gfCNCPoint1[3633] = {X 302.1122, Y 47.7433, Z -1.3333, A 0.000, B 0.000, C 0.000 }
gfCNCPoint1[3634] = {X 301.5880, Y 46.9091, Z -1.3333, A 0.000, B 0.000, C 0.000 }
gfCNCPoint1[3635] = {X 301.2626, Y 45.9790, Z -1.3333, A 0.000, B 0.000, C 0.000 }
gfCNCPoint1[3636] = {X 301.1523, Y 44.9999, Z -1.3333, A 0.000, B 0.000, C 0.000 }
gfCNCPoint1[3637] = {X 301.1524, Y 44.1991, Z -1.3333, A 0.000, B 0.000, C 0.000 }
gfCNCPoint1[3638] = {X 301.2707, Y 43.2557, Z -1.3333, A 0.000, B 0.000, C 0.000 }
gfCNCPoint1[3639] = {X 301.5741, Y 42.3546, Z -1.3333, A 0.000, B 0.000, C 0.000 }
gfCNCPoint1[3640] = {X 302.0506, Y 41.5318, Z -1.3333, A 0.000, B 0.000, C 0.000 }
gfCNCPoint1[3641] = {X 302.6811, Y 40.8202, Z -1.3333, A 0.000, B 0.000, C 0.000 }
gfCNCPoint1[3642] = {X 302.6811, Y 34.1143, Z -1.3333, A 0.000, B 0.000, C 0.000 }
gfCNCPoint1[3643] = {X 293.9335, Y 34.1143, Z -1.3333, A 0.000, B 0.000, C 0.000 }
gfCNCPoint1[3644] = {X 293.9325, Y 40.8666, Z -1.3333, A 0.000, B 0.000, C 0.000 }
gfCNCPoint1[3645] = {X 294.5724, Y 41.5615, Z -1.3333, A 0.000, B 0.000, C 0.000 }
gfCNCPoint1[3646] = {X 295.0533, Y 42.3747, Z -1.3333, A 0.000, B 0.000, C 0.000 }
gfCNCPoint1[3647] = {X 295.3539, Y 43.2703, Z -1.3333, A 0.000, B 0.000, C 0.000 }
gfCNCPoint1[3648] = {X 295.4611, Y 44.2089, Z -1.3333, A 0.000, B 0.000, C 0.000 }
gfCNCPoint1[3649] = {X 295.4611, Y 45.0000, Z -1.3333, A 0.000, B 0.000, C 0.000 }
gfCNCPoint1[3650] = {X 295.3508, Y 45.9791, Z -1.3333, A 0.000, B 0.000, C 0.000 }
gfCNCPoint1[3651] = {X 295.0254, Y 46.9091, Z -1.3333, A 0.000, B 0.000, C 0.000 }
gfCNCPoint1[3652] = {X 294.5012, Y 47.7434, Z -1.3333, A 0.000, B 0.000, C 0.000 }
gfCNCPoint1[3653] = {X 293.8045, Y 48.4401, Z -1.3333, A 0.000, B 0.000, C 0.000 }
gfCNCPoint1[3654] = {X 292.9702, Y 48.9643, Z -1.3333, A 0.000, B 0.000, C 0.000 }
gfCNCPoint1[3655] = {X 292.0402, Y 49.2897, Z -1.3333, A 0.000, B 0.000, C 0.000 }
gfCNCPoint1[3656] = {X 291.0611, Y 49.4000, Z -1.3333, A 0.000, B 0.000, C 0.000 }
gfCNCPoint1[3657] = {X 284.6177, Y 49.4000, Z -1.3333, A 0.000, B 0.000, C 0.000 }
gfCNCPoint1[3658] = {X 283.6386, Y 49.2897, Z -1.3333, A 0.000, B 0.000, C 0.000 }
gfCNCPoint1[3659] = {X 282.7086, Y 48.9643, Z -1.3333, A 0.000, B 0.000, C 0.000 }
gfCNCPoint1[3660] = {X 281.8743, Y 48.4400, Z -1.3333, A 0.000, B 0.000, C 0.000 }
gfCNCPoint1[3661] = {X 281.1776, Y 47.7433, Z -1.3333, A 0.000, B 0.000, C 0.000 }
gfCNCPoint1[3662] = {X 280.6534, Y 46.9091, Z -1.3333, A 0.000, B 0.000, C 0.000 }
gfCNCPoint1[3663] = {X 280.3280, Y 45.9791, Z -1.3333, A 0.000, B 0.000, C 0.000 }
gfCNCPoint1[3664] = {X 280.2177, Y 45.0000, Z -1.3333, A 0.000, B 0.000, C 0.000 }
gfCNCPoint1[3665] = {X 280.2177, Y 44.2065, Z -1.3333, A 0.000, B 0.000, C 0.000 }
gfCNCPoint1[3666] = {X 280.3232, Y 43.2697, Z -1.3333, A 0.000, B 0.000, C 0.000 }
gfCNCPoint1[3667] = {X 280.6235, Y 42.3761, Z -1.3333, A 0.000, B 0.000, C 0.000 }
gfCNCPoint1[3668] = {X 281.1051, Y 41.5657, Z -1.3333, A 0.000, B 0.000, C 0.000 }
gfCNCPoint1[3669] = {X 281.7465, Y 40.8749, Z -1.3333, A 0.000, B 0.000, C 0.000 }
gfCNCPoint1[3670] = {X 281.7461, Y 16.3118, Z -1.3333, A 0.000, B 0.000, C 0.000 }
gfCNCPoint1[3671] = {X 281.1011, Y 15.6226, Z -1.3333, A 0.000, B 0.000, C 0.000 }
gfCNCPoint1[3672] = {X 280.6180, Y 14.8117, Z -1.3333, A 0.000, B 0.000, C 0.000 }
gfCNCPoint1[3673] = {X 280.3189, Y 13.9164, Z -1.3333, A 0.000, B 0.000, C 0.000 }
gfCNCPoint1[3674] = {X 280.2177, Y 12.9779, Z -1.3333, A 0.000, B 0.000, C 0.000 }
gfCNCPoint1[3675] = {X 280.2177, Y 12.1868, Z -1.3333, A 0.000, B 0.000, C 0.000 }
gfCNCPoint1[3676] = {X 280.3280, Y 11.2077, Z -1.3333, A 0.000, B 0.000, C 0.000 }
gfCNCPoint1[3677] = {X 280.6534, Y 10.2777, Z -1.3333, A 0.000, B 0.000, C 0.000 }
gfCNCPoint1[3678] = {X 281.1776, Y 9.4435, Z -1.3333, A 0.000, B 0.000, C 0.000 }
gfCNCPoint1[3679] = {X 281.8743, Y 8.7468, Z -1.3333, A 0.000, B 0.000, C 0.000 }
gfCNCPoint1[3680] = {X 282.7086, Y 8.2226, Z -1.3333, A 0.000, B 0.000, C 0.000 }
gfCNCPoint1[3681] = {X 283.6386, Y 7.8971, Z -1.3333, A 0.000, B 0.000, C 0.000 }
gfCNCPoint1[3682] = {X 284.6177, Y 7.7868, Z -1.3333, A 0.000, B 0.000, C 0.000 }
gfCNCPoint1[3683] = {X 291.0611, Y 7.7868, Z -1.3333, A 0.000, B 0.000, C 0.000 }
gfCNCPoint1[3684] = {X 292.0402, Y 7.8971, Z -1.3333, A 0.000, B 0.000, C 0.000 }
gfCNCPoint1[3685] = {X 292.9702, Y 8.2226, Z -1.3333, A 0.000, B 0.000, C 0.000 }
gfCNCPoint1[3686] = {X 293.8045, Y 8.7468, Z -1.3333, A 0.000, B 0.000, C 0.000 }
gfCNCPoint1[3687] = {X 294.5012, Y 9.4435, Z -1.3333, A 0.000, B 0.000, C 0.000 }
gfCNCPoint1[3688] = {X 295.0254, Y 10.2777, Z -1.3333, A 0.000, B 0.000, C 0.000 }
gfCNCPoint1[3689] = {X 295.3508, Y 11.2077, Z -1.3333, A 0.000, B 0.000, C 0.000 }
gfCNCPoint1[3690] = {X 295.4611, Y 12.1868, Z -1.3333, A 0.000, B 0.000, C 0.000 }
gfCNCPoint1[3691] = {X 295.4609, Y 13.0233, Z -1.3333, A 0.000, B 0.000, C 0.000 }
gfCNCPoint1[3692] = {X 295.3525, Y 13.9497, Z -1.3333, A 0.000, B 0.000, C 0.000 }
gfCNCPoint1[3693] = {X 295.0512, Y 14.8325, Z -1.3333, A 0.000, B 0.000, C 0.000 }
gfCNCPoint1[3694] = {X 294.5707, Y 15.6319, Z -1.3333, A 0.000, B 0.000, C 0.000 }
gfCNCPoint1[3695] = {X 293.9324, Y 16.3121, Z -1.3333, A 0.000, B 0.000, C 0.000 }
gfCNCPoint1[3696] = {X 293.9337, Y 22.1165, Z -1.3333, A 0.000, B 0.000, C 0.000 }
gfCNCPoint1[3697] = {X 302.6799, Y 22.1165, Z -1.3333, A 0.000, B 0.000, C 0.000 }
gfCNCPoint1[3698] = {X 302.6806, Y 16.3117, Z -1.3333, A 0.000, B 0.000, C 0.000 }
gfCNCPoint1[3699] = {X 302.0356, Y 15.6225, Z -1.3333, A 0.000, B 0.000, C 0.000 }
gfCNCPoint1[3700] = {X 301.5525, Y 14.8116, Z -1.3333, A 0.000, B 0.000, C 0.000 }
gfCNCPoint1[3701] = {X 301.2535, Y 13.9164, Z -1.3333, A 0.000, B 0.000, C 0.000 }
gfCNCPoint1[3702] = {X 301.1523, Y 12.9779, Z -1.3333, A 0.000, B 0.000, C 0.000 }
gfCNCPoint1[3703] = {X 301.1523, Y 12.1868, Z -1.3333, A 0.000, B 0.000, C 0.000 }
gfCNCPoint1[3704] = {X 301.2626, Y 11.2077, Z -1.3333, A 0.000, B 0.000, C 0.000 }
gfCNCPoint1[3705] = {X 301.5880, Y 10.2777, Z -1.3333, A 0.000, B 0.000, C 0.000 }
gfCNCPoint1[3706] = {X 302.1122, Y 9.4435, Z -1.3333, A 0.000, B 0.000, C 0.000 }
gfCNCPoint1[3707] = {X 302.8089, Y 8.7468, Z -1.3333, A 0.000, B 0.000, C 0.000 }
gfCNCPoint1[3708] = {X 303.6432, Y 8.2226, Z -1.3333, A 0.000, B 0.000, C 0.000 }
gfCNCPoint1[3709] = {X 304.5732, Y 7.8971, Z -1.3333, A 0.000, B 0.000, C 0.000 }
gfCNCPoint1[3710] = {X 305.5523, Y 7.7868, Z -1.3333, A 0.000, B 0.000, C 0.000 }
gfCNCPoint1[3711] = {X 311.9957, Y 7.7868, Z -1.3333, A 0.000, B 0.000, C 0.000 }
gfCNCPoint1[3712] = {X 312.9748, Y 7.8971, Z -1.3333, A 0.000, B 0.000, C 0.000 }
gfCNCPoint1[3713] = {X 313.9048, Y 8.2226, Z -1.3333, A 0.000, B 0.000, C 0.000 }
gfCNCPoint1[3714] = {X 314.7391, Y 8.7468, Z -1.3333, A 0.000, B 0.000, C 0.000 }
gfCNCPoint1[3715] = {X 315.4358, Y 9.4435, Z -1.3333, A 0.000, B 0.000, C 0.000 }
gfCNCPoint1[3716] = {X 315.9600, Y 10.2777, Z -1.3333, A 0.000, B 0.000, C 0.000 }
gfCNCPoint1[3717] = {X 316.2854, Y 11.2077, Z -1.3333, A 0.000, B 0.000, C 0.000 }
gfCNCPoint1[3718] = {X 316.3957, Y 12.1868, Z -1.3333, A 0.000, B 0.000, C 0.000 }
gfCNCPoint1[3719] = {X 316.3955, Y 13.0233, Z -1.3333, A 0.000, B 0.000, C 0.000 }
gfCNCPoint1[3720] = {X 316.2871, Y 13.9497, Z -1.3333, A 0.000, B 0.000, C 0.000 }
gfCNCPoint1[3721] = {X 315.9859, Y 14.8324, Z -1.3333, A 0.000, B 0.000, C 0.000 }
gfCNCPoint1[3722] = {X 315.5054, Y 15.6318, Z -1.3333, A 0.000, B 0.000, C 0.000 }
gfCNCPoint1[3723] = {X 314.8671, Y 16.3119, Z -1.3333, A 0.000, B 0.000, C 0.000 }
gfCNCPoint1[3724] = {X 314.8669, Y 40.8747, Z -1.3333, A 0.000, B 0.000, C 0.000 }
gfCNCPoint1[3725] = {X 315.5120, Y 41.5639, Z -1.3333, A 0.000, B 0.000, C 0.000 }
gfCNCPoint1[3726] = {X 315.9953, Y 42.3749, Z -1.3333, A 0.000, B 0.000, C 0.000 }
gfCNCPoint1[3727] = {X 316.2945, Y 43.2703, Z -1.3333, A 0.000, B 0.000, C 0.000 }
gfCNCPoint1[3728] = {X 316.3957, Y 44.2089, Z -1.3333, A 0.000, B 0.000, C 0.000 }
gfCNCPoint1[3729] = {X 316.3957, Y 45.0000, Z -1.3333, A 0.000, B 0.000, C 0.000 }
gfCNCPoint1[3730] = {X 316.3190, Y 45.8182, Z -1.3333, A 0.000, B 0.000, C 0.000 }
gfCNCPoint1[3731] = {X 316.0914, Y 46.6079, Z -1.3333, A 0.000, B 0.000, C 0.000 }
gfCNCPoint1[3732] = {X 315.7209, Y 47.3415, Z -1.3333, A 0.000, B 0.000, C 0.000 }
gfCNCPoint1[3733] = {X 315.2205, Y 47.9934, Z -1.3333, A 0.000, B 0.000, C 0.000 }
gfCNCPoint1[3734] = {X 315.5723, Y 48.3200, Z -1.3333, A 0.000, B 0.000, C 0.000 }
gfCNCPoint1[3735] = {X 324.3107, Y 48.3200, Z -1.3333, A 0.000, B 0.000, C 0.000 }
gfCNCPoint1[3736] = {X 325.5555, Y 48.4004, Z -1.3333, A 0.000, B 0.000, C 0.000 }
gfCNCPoint1[3737] = {X 326.7797, Y 48.6402, Z -1.3333, A 0.000, B 0.000, C 0.000 }
gfCNCPoint1[3738] = {X 325.5882, Y 48.0963, Z -1.3333, A 0.000, B 0.000, C 0.000 }
gfCNCPoint1[3739] = {X 324.4810, Y 47.3966, Z -1.3333, A 0.000, B 0.000, C 0.000 }
gfCNCPoint1[3740] = {X 323.4784, Y 46.5538, Z -1.3333, A 0.000, B 0.000, C 0.000 }
gfCNCPoint1[3741] = {X 322.8382, Y 45.9295, Z -1.3333, A 0.000, B 0.000, C 0.000 }
gfCNCPoint1[3742] = {X 322.2180, Y 45.2650, Z -1.3333, A 0.000, B 0.000, C 0.000 }
gfCNCPoint1[3743] = {X 321.6628, Y 44.5452, Z -1.3333, A 0.000, B 0.000, C 0.000 }
gfCNCPoint1[3744] = {X 323.6300, Y 43.1703, Z -1.3333, A 0.000, B 0.000, C 0.000 }
gfCNCPoint1[3745] = {X 323.0063, Y 42.0918, Z -1.3333, A 0.000, B 0.000, C 0.000 }
gfCNCPoint1[3746] = {X 322.5757, Y 40.9227, Z -1.3333, A 0.000, B 0.000, C 0.000 }
gfCNCPoint1[3747] = {X 322.3506, Y 39.6973, Z -1.3333, A 0.000, B 0.000, C 0.000 }
gfCNCPoint1[3748] = {X 322.3379, Y 38.4514, Z -1.3333, A 0.000, B 0.000, C 0.000 }
gfCNCPoint1[3749] = {X 322.5377, Y 37.2217, Z -1.3333, A 0.000, B 0.000, C 0.000 }
gfCNCPoint1[3750] = {X 322.9443, Y 36.0440, Z -1.3333, A 0.000, B 0.000, C 0.000 }
gfCNCPoint1[3751] = {X 323.5458, Y 34.9529, Z -1.3333, A 0.000, B 0.000, C 0.000 }
gfCNCPoint1[3752] = {X 327.7789, Y 28.6234, Z -1.3333, A 0.000, B 0.000, C 0.000 }
gfCNCPoint1[3753] = {X 328.5158, Y 27.6951, Z -1.3333, A 0.000, B 0.000, C 0.000 }
gfCNCPoint1[3754] = {X 329.3935, Y 26.8986, Z -1.3333, A 0.000, B 0.000, C 0.000 }
gfCNCPoint1[3755] = {X 330.3889, Y 26.2552, Z -1.3333, A 0.000, B 0.000, C 0.000 }
gfCNCPoint1[3756] = {X 331.5063, Y 25.7713, Z -1.3333, A 0.000, B 0.000, C 0.000 }
gfCNCPoint1[3757] = {X 332.6887, Y 25.4804, Z -1.3333, A 0.000, B 0.000, C 0.000 }
gfCNCPoint1[3758] = {X 333.9031, Y 25.3907, Z -1.3333, A 0.000, B 0.000, C 0.000 }
gfCNCPoint1[3759] = {X 335.1154, Y 25.5046, Z -1.3333, A 0.000, B 0.000, C 0.000 }
gfCNCPoint1[3760] = {X 336.2918, Y 25.8191, Z -1.3333, A 0.000, B 0.000, C 0.000 }
gfCNCPoint1[3761] = {X 337.3993, Y 26.3252, Z -1.3333, A 0.000, B 0.000, C 0.000 }
gfCNCPoint1[3762] = {X 338.1754, Y 26.8292, Z -1.3333, A 0.000, B 0.000, C 0.000 }
gfCNCPoint1[3763] = {X 338.8813, Y 27.4275, Z -1.3333, A 0.000, B 0.000, C 0.000 }
gfCNCPoint1[3764] = {X 339.5028, Y 28.0267, Z -1.3333, A 0.000, B 0.000, C 0.000 }
gfCNCPoint1[3765] = {X 340.3316, Y 28.9979, Z -1.3333, A 0.000, B 0.000, C 0.000 }
gfCNCPoint1[3766] = {X 340.9780, Y 30.0990, Z -1.3333, A 0.000, B 0.000, C 0.000 }
gfCNCPoint1[3767] = {X 341.4220, Y 31.2960, Z -1.3333, A 0.000, B 0.000, C 0.000 }
gfCNCPoint1[3768] = {X 341.6501, Y 32.5522, Z -1.3333, A 0.000, B 0.000, C 0.000 }
gfCNCPoint1[3769] = {X 341.8439, Y 32.7095, Z -1.3333, A 0.000, B 0.000, C 0.000 }
gfCNCPoint1[3770] = {X 342.0399, Y 32.8640, Z -1.3333, A 0.000, B 0.000, C 0.000 }
gfCNCPoint1[3771] = {X 342.9828, Y 33.4816, Z -1.3333, A 0.000, B 0.000, C 0.000 }
gfCNCPoint1[3772] = {X 344.0063, Y 33.9541, Z -1.3333, A 0.000, B 0.000, C 0.000 }
gfCNCPoint1[3773] = {X 345.0879, Y 34.2712, Z -1.3333, A 0.000, B 0.000, C 0.000 }
gfCNCPoint1[3774] = {X 346.2045, Y 34.4260, Z -1.3333, A 0.000, B 0.000, C 0.000 }
gfCNCPoint1[3775] = {X 347.3316, Y 34.4151, Z -1.3333, A 0.000, B 0.000, C 0.000 }
gfCNCPoint1[3776] = {X 348.3037, Y 34.2892, Z -1.3333, A 0.000, B 0.000, C 0.000 }
gfCNCPoint1[3777] = {X 349.2417, Y 34.0051, Z -1.3333, A 0.000, B 0.000, C 0.000 }
gfCNCPoint1[3778] = {X 350.1202, Y 33.5705, Z -1.3333, A 0.000, B 0.000, C 0.000 }
gfCNCPoint1[3779] = {X 350.9153, Y 32.9973, Z -1.3333, A 0.000, B 0.000, C 0.000 }
gfCNCPoint1[3780] = {X 351.7896, Y 32.1460, Z -1.3333, A 0.000, B 0.000, C 0.000 }
gfCNCPoint1[3781] = {X 352.5466, Y 31.1888, Z -1.3333, A 0.000, B 0.000, C 0.000 }
gfCNCPoint1[3782] = {X 353.1735, Y 30.1418, Z -1.3333, A 0.000, B 0.000, C 0.000 }
gfCNCPoint1[3783] = {X 353.6598, Y 29.0226, Z -1.3333, A 0.000, B 0.000, C 0.000 }
gfCNCPoint1[3784] = {X 353.9974, Y 27.8499, Z -1.3333, A 0.000, B 0.000, C 0.000 }
gfCNCPoint1[3785] = {X 354.2247, Y 26.4401, Z -1.3333, A 0.000, B 0.000, C 0.000 }
gfCNCPoint1[3786] = {X 354.3167, Y 25.0152, Z -1.3333, A 0.000, B 0.000, C 0.000 }
gfCNCPoint1[3787] = {X 354.2727, Y 23.5879, Z -1.3333, A 0.000, B 0.000, C 0.000 }
gfCNCPoint1[3788] = {X 354.0929, Y 22.1713, Z -1.3333, A 0.000, B 0.000, C 0.000 }
gfCNCPoint1[3789] = {X 353.8402, Y 21.0759, Z -1.3333, A 0.000, B 0.000, C 0.000 }
gfCNCPoint1[3790] = {X 353.4535, Y 20.0203, Z -1.3333, A 0.000, B 0.000, C 0.000 }
gfCNCPoint1[3791] = {X 352.9388, Y 19.0209, Z -1.3333, A 0.000, B 0.000, C 0.000 }
gfCNCPoint1[3792] = {X 352.3040, Y 18.0930, Z -1.3333, A 0.000, B 0.000, C 0.000 }
gfCNCPoint1[3793] = {X 351.5370, Y 17.2656, Z -1.3333, A 0.000, B 0.000, C 0.000 }
gfCNCPoint1[3794] = {X 350.6343, Y 16.5887, Z -1.3333, A 0.000, B 0.000, C 0.000 }
gfCNCPoint1[3795] = {X 349.6251, Y 16.0843, Z -1.3333, A 0.000, B 0.000, C 0.000 }
gfCNCPoint1[3796] = {X 348.5419, Y 15.7685, Z -1.3333, A 0.000, B 0.000, C 0.000 }
gfCNCPoint1[3797] = {X 347.1562, Y 15.5979, Z -1.3333, A 0.000, B 0.000, C 0.000 }
gfCNCPoint1[3798] = {X 345.7602, Y 15.6140, Z -1.3333, A 0.000, B 0.000, C 0.000 }
gfCNCPoint1[3799] = {X 344.3788, Y 15.8165, Z -1.3333, A 0.000, B 0.000, C 0.000 }
gfCNCPoint1[3800] = {X 343.0368, Y 16.2017, Z -1.3333, A 0.000, B 0.000, C 0.000 }
gfCNCPoint1[3801] = {X 341.7584, Y 16.7629, Z -1.3333, A 0.000, B 0.000, C 0.000 }
gfCNCPoint1[3802] = {X 341.4307, Y 17.8582, Z -1.3333, A 0.000, B 0.000, C 0.000 }
gfCNCPoint1[3803] = {X 340.9356, Y 18.8888, Z -1.3333, A 0.000, B 0.000, C 0.000 }
gfCNCPoint1[3804] = {X 340.2853, Y 19.8292, Z -1.3333, A 0.000, B 0.000, C 0.000 }
gfCNCPoint1[3805] = {X 345.8671, Y 24.3770, Z -1.3333, A 0.000, B 0.000, C 0.000 }
gfCNCPoint1[3806] = {X 346.4664, Y 25.2140, Z -1.3333, A 0.000, B 0.000, C 0.000 }
gfCNCPoint1[3807] = {X 347.0046, Y 26.0914, Z -1.3333, A 0.000, B 0.000, C 0.000 }
gfCNCPoint1[3808] = {X 347.1188, Y 24.7351, Z -1.3333, A 0.000, B 0.000, C 0.000 }
gfCNCPoint1[3809] = {X 346.9949, Y 23.3798, Z -1.3333, A 0.000, B 0.000, C 0.000 }
gfCNCPoint1[3810] = {X 346.9507, Y 23.1695, Z -1.3333, A 0.000, B 0.000, C 0.000 }
gfCNCPoint1[3811] = {X 346.8823, Y 22.9658, Z -1.3333, A 0.000, B 0.000, C 0.000 }
gfCNCPoint1[3812] = {X 346.3959, Y 23.6867, Z -1.3333, A 0.000, B 0.000, C 0.000 }
gfCNCPoint1[3813] = {X 345.8671, Y 24.3770, Z -1.3333, A 0.000, B 0.000, C 0.000 }
gfCNCPoint1[3814] = {X 344.0065, Y 22.8611, Z -1.3333, A 0.000, B 0.000, C 0.000 }
gfCNCPoint1[3815] = {X 343.3271, Y 23.6263, Z -1.3333, A 0.000, B 0.000, C 0.000 }
gfCNCPoint1[3816] = {X 342.5854, Y 24.3313, Z -1.3333, A 0.000, B 0.000, C 0.000 }
gfCNCPoint1[3817] = {X 342.8589, Y 24.5949, Z -1.3333, A 0.000, B 0.000, C 0.000 }
gfCNCPoint1[3818] = {X 343.9812, Y 25.8617, Z -1.3333, A 0.000, B 0.000, C 0.000 }
gfCNCPoint1[3819] = {X 344.9156, Y 27.2729, Z -1.3333, A 0.000, B 0.000, C 0.000 }
gfCNCPoint1[3820] = {X 345.4672, Y 28.3762, Z -1.3333, A 0.000, B 0.000, C 0.000 }
gfCNCPoint1[3821] = {X 345.9035, Y 29.5300, Z -1.3333, A 0.000, B 0.000, C 0.000 }
gfCNCPoint1[3822] = {X 346.4600, Y 29.6326, Z -1.3333, A 0.000, B 0.000, C 0.000 }
gfCNCPoint1[3823] = {X 347.0258, Y 29.6235, Z -1.3333, A 0.000, B 0.000, C 0.000 }
gfCNCPoint1[3824] = {X 347.4365, Y 29.5578, Z -1.3333, A 0.000, B 0.000, C 0.000 }
gfCNCPoint1[3825] = {X 347.7961, Y 29.3489, Z -1.3333, A 0.000, B 0.000, C 0.000 }
gfCNCPoint1[3826] = {X 348.4760, Y 28.6282, Z -1.3333, A 0.000, B 0.000, C 0.000 }
gfCNCPoint1[3827] = {X 348.9866, Y 27.7791, Z -1.3333, A 0.000, B 0.000, C 0.000 }
gfCNCPoint1[3828] = {X 349.3046, Y 26.8407, Z -1.3333, A 0.000, B 0.000, C 0.000 }
gfCNCPoint1[3829] = {X 349.3384, Y 26.6711, Z -1.3333, A 0.000, B 0.000, C 0.000 }
gfCNCPoint1[3830] = {X 349.3694, Y 26.5010, Z -1.3333, A 0.000, B 0.000, C 0.000 }
gfCNCPoint1[3831] = {X 349.5031, Y 25.3293, Z -1.3333, A 0.000, B 0.000, C 0.000 }
gfCNCPoint1[3832] = {X 349.5003, Y 24.1499, Z -1.3333, A 0.000, B 0.000, C 0.000 }
gfCNCPoint1[3833] = {X 349.3613, Y 22.9788, Z -1.3333, A 0.000, B 0.000, C 0.000 }
gfCNCPoint1[3834] = {X 349.1892, Y 22.2869, Z -1.3333, A 0.000, B 0.000, C 0.000 }
gfCNCPoint1[3835] = {X 348.9038, Y 21.6335, Z -1.3333, A 0.000, B 0.000, C 0.000 }
gfCNCPoint1[3836] = {X 348.5130, Y 21.0371, Z -1.3333, A 0.000, B 0.000, C 0.000 }
gfCNCPoint1[3837] = {X 348.1202, Y 20.6777, Z -1.3333, A 0.000, B 0.000, C 0.000 }
gfCNCPoint1[3838] = {X 347.6258, Y 20.4803, Z -1.3333, A 0.000, B 0.000, C 0.000 }
gfCNCPoint1[3839] = {X 346.5729, Y 20.3819, Z -1.3333, A 0.000, B 0.000, C 0.000 }
gfCNCPoint1[3840] = {X 345.5203, Y 20.4822, Z -1.3333, A 0.000, B 0.000, C 0.000 }
gfCNCPoint1[3841] = {X 344.8330, Y 21.7160, Z -1.3333, A 0.000, B 0.000, C 0.000 }
gfCNCPoint1[3842] = {X 344.0065, Y 22.8611, Z -1.3333, A 0.000, B 0.000, C 0.000 }
gfCNCPoint1[3843] = {X 342.1459, Y 21.3451, Z -1.3333, A 0.000, B 0.000, C 0.000 }
gfCNCPoint1[3844] = {X 341.6015, Y 21.9583, Z -1.3333, A 0.000, B 0.000, C 0.000 }
gfCNCPoint1[3845] = {X 341.0072, Y 22.5232, Z -1.3333, A 0.000, B 0.000, C 0.000 }
gfCNCPoint1[3846] = {X 340.7216, Y 22.7630, Z -1.3333, A 0.000, B 0.000, C 0.000 }
gfCNCPoint1[3847] = {X 340.4270, Y 22.9916, Z -1.3333, A 0.000, B 0.000, C 0.000 }
gfCNCPoint1[3848] = {X 339.6615, Y 23.5549, Z -1.3333, A 0.000, B 0.000, C 0.000 }
gfCNCPoint1[3849] = {X 339.1299, Y 23.9121, Z -1.3333, A 0.000, B 0.000, C 0.000 }
gfCNCPoint1[3850] = {X 338.5759, Y 24.2333, Z -1.3333, A 0.000, B 0.000, C 0.000 }
gfCNCPoint1[3851] = {X 339.6079, Y 24.9035, Z -1.3333, A 0.000, B 0.000, C 0.000 }
gfCNCPoint1[3852] = {X 340.5465, Y 25.6991, Z -1.3333, A 0.000, B 0.000, C 0.000 }
gfCNCPoint1[3853] = {X 341.1848, Y 26.3148, Z -1.3333, A 0.000, B 0.000, C 0.000 }
gfCNCPoint1[3854] = {X 342.1202, Y 27.3792, Z -1.3333, A 0.000, B 0.000, C 0.000 }
gfCNCPoint1[3855] = {X 342.8902, Y 28.5687, Z -1.3333, A 0.000, B 0.000, C 0.000 }
gfCNCPoint1[3856] = {X 343.4783, Y 29.8579, Z -1.3333, A 0.000, B 0.000, C 0.000 }
gfCNCPoint1[3857] = {X 343.8718, Y 31.2192, Z -1.3333, A 0.000, B 0.000, C 0.000 }
gfCNCPoint1[3858] = {X 344.6368, Y 31.6221, Z -1.3333, A 0.000, B 0.000, C 0.000 }
gfCNCPoint1[3859] = {X 345.4575, Y 31.8941, Z -1.3333, A 0.000, B 0.000, C 0.000 }
gfCNCPoint1[3860] = {X 346.3117, Y 32.0279, Z -1.3333, A 0.000, B 0.000, C 0.000 }
gfCNCPoint1[3861] = {X 347.1763, Y 32.0198, Z -1.3333, A 0.000, B 0.000, C 0.000 }
gfCNCPoint1[3862] = {X 347.9605, Y 31.9045, Z -1.3333, A 0.000, B 0.000, C 0.000 }
gfCNCPoint1[3863] = {X 348.6994, Y 31.6174, Z -1.3333, A 0.000, B 0.000, C 0.000 }
gfCNCPoint1[3864] = {X 349.3558, Y 31.1730, Z -1.3333, A 0.000, B 0.000, C 0.000 }
gfCNCPoint1[3865] = {X 350.1556, Y 30.3689, Z -1.3333, A 0.000, B 0.000, C 0.000 }
gfCNCPoint1[3866] = {X 350.8155, Y 29.4466, Z -1.3333, A 0.000, B 0.000, C 0.000 }
gfCNCPoint1[3867] = {X 351.3183, Y 28.4300, Z -1.3333, A 0.000, B 0.000, C 0.000 }
gfCNCPoint1[3868] = {X 351.6509, Y 27.3457, Z -1.3333, A 0.000, B 0.000, C 0.000 }
gfCNCPoint1[3869] = {X 351.8790, Y 25.7632, Z -1.3333, A 0.000, B 0.000, C 0.000 }
gfCNCPoint1[3870] = {X 351.9046, Y 24.1645, Z -1.3333, A 0.000, B 0.000, C 0.000 }
gfCNCPoint1[3871] = {X 351.7272, Y 22.5755, Z -1.3333, A 0.000, B 0.000, C 0.000 }
gfCNCPoint1[3872] = {X 351.4581, Y 21.5045, Z -1.3333, A 0.000, B 0.000, C 0.000 }
gfCNCPoint1[3873] = {X 351.0154, Y 20.4929, Z -1.3333, A 0.000, B 0.000, C 0.000 }
gfCNCPoint1[3874] = {X 350.4112, Y 19.5685, Z -1.3333, A 0.000, B 0.000, C 0.000 }
gfCNCPoint1[3875] = {X 349.7601, Y 18.9037, Z -1.3333, A 0.000, B 0.000, C 0.000 }
gfCNCPoint1[3876] = {X 348.9693, Y 18.4129, Z -1.3333, A 0.000, B 0.000, C 0.000 }
gfCNCPoint1[3877] = {X 348.0845, Y 18.1246, Z -1.3333, A 0.000, B 0.000, C 0.000 }
gfCNCPoint1[3878] = {X 346.9931, Y 17.9926, Z -1.3333, A 0.000, B 0.000, C 0.000 }
gfCNCPoint1[3879] = {X 345.8939, Y 18.0111, Z -1.3333, A 0.000, B 0.000, C 0.000 }
gfCNCPoint1[3880] = {X 344.8076, Y 18.1796, Z -1.3333, A 0.000, B 0.000, C 0.000 }
gfCNCPoint1[3881] = {X 343.7545, Y 18.4950, Z -1.3333, A 0.000, B 0.000, C 0.000 }
gfCNCPoint1[3882] = {X 343.3272, Y 19.5038, Z -1.3333, A 0.000, B 0.000, C 0.000 }
gfCNCPoint1[3883] = {X 342.7888, Y 20.4580, Z -1.3333, A 0.000, B 0.000, C 0.000 }
gfCNCPoint1[3884] = {X 342.1459, Y 21.3451, Z -1.3333, A 0.000, B 0.000, C 0.000 }
gfCNCPoint1[3885] = {X 340.2853, Y 19.8292, Z -1.3333, A 0.000, B 0.000, C 0.000 }
gfCNCPoint1[3886] = {X 339.6794, Y 20.4860, Z -1.3333, A 0.000, B 0.000, C 0.000 }
gfCNCPoint1[3887] = {X 338.9976, Y 21.0636, Z -1.3333, A 0.000, B 0.000, C 0.000 }
gfCNCPoint1[3888] = {X 338.2497, Y 21.6140, Z -1.3333, A 0.000, B 0.000, C 0.000 }
gfCNCPoint1[3889] = {X 337.8538, Y 21.8795, Z -1.3333, A 0.000, B 0.000, C 0.000 }
gfCNCPoint1[3890] = {X 337.4413, Y 22.1185, Z -1.3333, A 0.000, B 0.000, C 0.000 }
gfCNCPoint1[3891] = {X 336.3239, Y 22.6023, Z -1.3333, A 0.000, B 0.000, C 0.000 }
gfCNCPoint1[3892] = {X 335.1415, Y 22.8932, Z -1.3333, A 0.000, B 0.000, C 0.000 }
gfCNCPoint1[3893] = {X 333.9271, Y 22.9829, Z -1.3333, A 0.000, B 0.000, C 0.000 }
gfCNCPoint1[3894] = {X 332.7148, Y 22.8690, Z -1.3333, A 0.000, B 0.000, C 0.000 }
gfCNCPoint1[3895] = {X 331.5384, Y 22.5546, Z -1.3333, A 0.000, B 0.000, C 0.000 }
gfCNCPoint1[3896] = {X 330.4309, Y 22.0485, Z -1.3333, A 0.000, B 0.000, C 0.000 }
gfCNCPoint1[3897] = {X 329.5143, Y 21.4374, Z -1.3333, A 0.000, B 0.000, C 0.000 }
gfCNCPoint1[3898] = {X 328.7005, Y 20.6949, Z -1.3333, A 0.000, B 0.000, C 0.000 }
gfCNCPoint1[3899] = {X 328.0080, Y 19.8382, Z -1.3333, A 0.000, B 0.000, C 0.000 }
gfCNCPoint1[3900] = {X 327.4527, Y 18.8868, Z -1.3333, A 0.000, B 0.000, C 0.000 }
gfCNCPoint1[3901] = {X 323.9321, Y 11.6443, Z -1.3333, A 0.000, B 0.000, C 0.000 }
gfCNCPoint1[3902] = {X 323.5337, Y 10.6422, Z -1.3333, A 0.000, B 0.000, C 0.000 }
gfCNCPoint1[3903] = {X 323.2878, Y 9.5922, Z -1.3333, A 0.000, B 0.000, C 0.000 }
gfCNCPoint1[3904] = {X 323.1997, Y 8.5174, Z -1.3333, A 0.000, B 0.000, C 0.000 }
gfCNCPoint1[3905] = {X 323.2713, Y 7.4414, Z -1.3333, A 0.000, B 0.000, C 0.000 }
gfCNCPoint1[3906] = {X 323.4719, Y 6.4885, Z -1.3333, A 0.000, B 0.000, C 0.000 }
gfCNCPoint1[3907] = {X 323.7979, Y 5.5710, Z -1.3333, A 0.000, B 0.000, C 0.000 }
gfCNCPoint1[3908] = {X 324.2435, Y 4.7051, Z -1.3333, A 0.000, B 0.000, C 0.000 }
gfCNCPoint1[3909] = {X 168.0205, Y 4.7051, Z -1.3333, A 0.000, B 0.000, C 0.000 }
gfCNCPoint1[3910] = {X 168.0205, Y 9.5051, Z -1.3333, A 0.000, B 0.000, C 0.000 }
gfCNCPoint1[3911] = {X 166.5360, Y 9.5051, Z -1.3333, A 0.000, B 0.000, C 0.000 }
gfCNCPoint1[3912] = {X 166.5856, Y 9.9932, Z -1.3333, A 0.000, B 0.000, C 0.000 }
gfCNCPoint1[3913] = {X 166.6021, Y 10.4835, Z -1.3333, A 0.000, B 0.000, C 0.000 }
gfCNCPoint1[3914] = {X 166.6021, Y 13.0969, Z -1.3333, A 0.000, B 0.000, C 0.000 }
gfCNCPoint1[3915] = {X 166.8569, Y 11.8210, Z -1.3333, A 0.000, B 0.000, C 0.000 }
gfCNCPoint1[3916] = {X 167.3348, Y 10.6109, Z -1.3333, A 0.000, B 0.000, C 0.000 }
gfCNCPoint1[3917] = {X 168.0205, Y 9.5051, Z -1.3333, A 0.000, B 0.000, C 0.000 }
gfCNCPoint1[3918] = {X 168.0205, Y 7.1051, Z -1.3333, A 0.000, B 0.000, C 0.000 }
gfCNCPoint1[3919] = {X 162.8436, Y 7.1051, Z -1.3333, A 0.000, B 0.000, C 0.000 }
gfCNCPoint1[3920] = {X 163.4703, Y 7.9132, Z -1.3333, A 0.000, B 0.000, C 0.000 }
gfCNCPoint1[3921] = {X 163.9149, Y 8.8342, Z -1.3333, A 0.000, B 0.000, C 0.000 }
gfCNCPoint1[3922] = {X 164.1578, Y 9.8277, Z -1.3333, A 0.000, B 0.000, C 0.000 }
gfCNCPoint1[3923] = {X 164.1910, Y 10.1548, Z -1.3333, A 0.000, B 0.000, C 0.000 }
gfCNCPoint1[3924] = {X 164.2021, Y 10.4835, Z -1.3333, A 0.000, B 0.000, C 0.000 }
gfCNCPoint1[3925] = {X 164.2021, Y 17.4615, Z -1.3333, A 0.000, B 0.000, C 0.000 }
gfCNCPoint1[3926] = {X 164.1140, Y 18.3848, Z -1.3333, A 0.000, B 0.000, C 0.000 }
gfCNCPoint1[3927] = {X 163.8527, Y 19.2747, Z -1.3333, A 0.000, B 0.000, C 0.000 }
gfCNCPoint1[3928] = {X 163.4279, Y 20.0991, Z -1.3333, A 0.000, B 0.000, C 0.000 }
gfCNCPoint1[3929] = {X 162.8547, Y 20.8282, Z -1.3333, A 0.000, B 0.000, C 0.000 }
gfCNCPoint1[3930] = {X 162.1540, Y 21.4358, Z -1.3333, A 0.000, B 0.000, C 0.000 }
gfCNCPoint1[3931] = {X 161.3510, Y 21.8998, Z -1.3333, A 0.000, B 0.000, C 0.000 }
gfCNCPoint1[3932] = {X 160.4746, Y 22.2035, Z -1.3333, A 0.000, B 0.000, C 0.000 }
gfCNCPoint1[3933] = {X 162.1751, Y 29.1998, Z -1.3333, A 0.000, B 0.000, C 0.000 }
gfCNCPoint1[3934] = {X 161.1121, Y 29.4082, Z -1.3333, A 0.000, B 0.000, C 0.000 }
gfCNCPoint1[3935] = {X 160.0347, Y 29.5205, Z -1.3333, A 0.000, B 0.000, C 0.000 }
gfCNCPoint1[3936] = {X 160.0340, Y 38.3367, Z -1.3333, A 0.000, B 0.000, C 0.000 }
gfCNCPoint1[3937] = {X 160.6822, Y 39.6937, Z -1.3333, A 0.000, B 0.000, C 0.000 }
gfCNCPoint1[3938] = {X 161.1574, Y 41.1206, Z -1.3333, A 0.000, B 0.000, C 0.000 }
gfCNCPoint1[3939] = {X 162.0490, Y 41.1205, Z -1.3333, A 0.000, B 0.000, C 0.000 }
gfCNCPoint1[3940] = {X 161.6748, Y 39.3712, Z -1.3333, A 0.000, B 0.000, C 0.000 }
gfCNCPoint1[3941] = {X 161.4508, Y 37.5963, Z -1.3333, A 0.000, B 0.000, C 0.000 }
gfCNCPoint1[3942] = {X 161.3323, Y 35.4809, Z -1.3333, A 0.000, B 0.000, C 0.000 }
gfCNCPoint1[3943] = {X 161.4144, Y 33.3637, Z -1.3333, A 0.000, B 0.000, C 0.000 }
gfCNCPoint1[3944] = {X 161.6961, Y 31.2637, Z -1.3333, A 0.000, B 0.000, C 0.000 }
gfCNCPoint1[3945] = {X 162.1751, Y 29.1998, Z -1.3333, A 0.000, B 0.000, C 0.000 }
gfCNCPoint1[3946] = {X 161.6083, Y 26.8677, Z -1.3333, A 0.000, B 0.000, C 0.000 }
gfCNCPoint1[3947] = {X 160.4733, Y 27.0728, Z -1.3333, A 0.000, B 0.000, C 0.000 }
gfCNCPoint1[3948] = {X 159.3220, Y 27.1415, Z -1.3333, A 0.000, B 0.000, C 0.000 }
gfCNCPoint1[3949] = {X 158.6670, Y 27.1415, Z -1.3333, A 0.000, B 0.000, C 0.000 }
gfCNCPoint1[3950] = {X 158.1502, Y 27.1259, Z -1.3333, A 0.000, B 0.000, C 0.000 }
gfCNCPoint1[3951] = {X 157.6349, Y 27.0829, Z -1.3333, A 0.000, B 0.000, C 0.000 }
gfCNCPoint1[3952] = {X 157.6339, Y 38.9962, Z -1.3333, A 0.000, B 0.000, C 0.000 }
gfCNCPoint1[3953] = {X 158.2178, Y 40.0485, Z -1.3333, A 0.000, B 0.000, C 0.000 }
gfCNCPoint1[3954] = {X 158.6672, Y 41.1650, Z -1.3333, A 0.000, B 0.000, C 0.000 }
gfCNCPoint1[3955] = {X 158.9752, Y 42.3284, Z -1.3333, A 0.000, B 0.000, C 0.000 }
gfCNCPoint1[3956] = {X 159.1372, Y 43.5209, Z -1.3333, A 0.000, B 0.000, C 0.000 }
gfCNCPoint1[3957] = {X 165.4308, Y 43.5200, Z -1.3333, A 0.000, B 0.000, C 0.000 }
gfCNCPoint1[3958] = {X 164.8373, Y 42.0421, Z -1.3333, A 0.000, B 0.000, C 0.000 }
gfCNCPoint1[3959] = {X 164.3724, Y 40.5189, Z -1.3333, A 0.000, B 0.000, C 0.000 }
gfCNCPoint1[3960] = {X 164.0389, Y 38.9575, Z -1.3333, A 0.000, B 0.000, C 0.000 }
gfCNCPoint1[3961] = {X 163.8406, Y 37.3733, Z -1.3333, A 0.000, B 0.000, C 0.000 }
gfCNCPoint1[3962] = {X 163.7324, Y 35.4786, Z -1.3333, A 0.000, B 0.000, C 0.000 }
gfCNCPoint1[3963] = {X 163.8044, Y 33.5822, Z -1.3333, A 0.000, B 0.000, C 0.000 }
gfCNCPoint1[3964] = {X 164.0559, Y 31.7011, Z -1.3333, A 0.000, B 0.000, C 0.000 }
gfCNCPoint1[3965] = {X 164.4847, Y 29.8524, Z -1.3333, A 0.000, B 0.000, C 0.000 }
gfCNCPoint1[3966] = {X 164.8366, Y 28.7335, Z -1.3333, A 0.000, B 0.000, C 0.000 }
gfCNCPoint1[3967] = {X 165.2535, Y 27.6373, Z -1.3333, A 0.000, B 0.000, C 0.000 }
gfCNCPoint1[3968] = {X 165.8702, Y 26.3065, Z -1.3333, A 0.000, B 0.000, C 0.000 }
gfCNCPoint1[3969] = {X 166.6046, Y 25.0369, Z -1.3333, A 0.000, B 0.000, C 0.000 }
gfCNCPoint1[3970] = {X 167.4506, Y 23.8388, Z -1.3333, A 0.000, B 0.000, C 0.000 }
gfCNCPoint1[3971] = {X 167.1640, Y 23.1367, Z -1.3333, A 0.000, B 0.000, C 0.000 }
gfCNCPoint1[3972] = {X 166.2874, Y 24.1837, Z -1.3333, A 0.000, B 0.000, C 0.000 }
gfCNCPoint1[3973] = {X 165.2722, Y 25.0969, Z -1.3333, A 0.000, B 0.000, C 0.000 }
gfCNCPoint1[3974] = {X 164.1386, Y 25.8582, Z -1.3333, A 0.000, B 0.000, C 0.000 }
gfCNCPoint1[3975] = {X 162.9091, Y 26.4524, Z -1.3333, A 0.000, B 0.000, C 0.000 }
gfCNCPoint1[3976] = {X 161.6083, Y 26.8677, Z -1.3333, A 0.000, B 0.000, C 0.000 }
gfCNCPoint1[3977] = {X 161.0415, Y 24.5356, Z -1.3333, A 0.000, B 0.000, C 0.000 }
gfCNCPoint1[3978] = {X 160.1879, Y 24.6899, Z -1.3333, A 0.000, B 0.000, C 0.000 }
gfCNCPoint1[3979] = {X 159.3220, Y 24.7415, Z -1.3333, A 0.000, B 0.000, C 0.000 }
gfCNCPoint1[3980] = {X 158.6755, Y 24.7415, Z -1.3333, A 0.000, B 0.000, C 0.000 }
gfCNCPoint1[3981] = {X 158.2863, Y 24.7298, Z -1.3333, A 0.000, B 0.000, C 0.000 }
gfCNCPoint1[3982] = {X 157.8982, Y 24.6974, Z -1.3333, A 0.000, B 0.000, C 0.000 }
gfCNCPoint1[3983] = {X 156.9776, Y 24.5357, Z -1.3333, A 0.000, B 0.000, C 0.000 }
gfCNCPoint1[3984] = {X 156.0851, Y 24.2580, Z -1.3333, A 0.000, B 0.000, C 0.000 }
gfCNCPoint1[3985] = {X 155.2352, Y 23.8689, Z -1.3333, A 0.000, B 0.000, C 0.000 }
gfCNCPoint1[3986] = {X 155.2339, Y 39.7517, Z -1.3333, A 0.000, B 0.000, C 0.000 }
gfCNCPoint1[3987] = {X 155.8247, Y 40.6440, Z -1.3333, A 0.000, B 0.000, C 0.000 }
gfCNCPoint1[3988] = {X 156.2792, Y 41.6127, Z -1.3333, A 0.000, B 0.000, C 0.000 }
gfCNCPoint1[3989] = {X 156.5877, Y 42.6374, Z -1.3333, A 0.000, B 0.000, C 0.000 }
gfCNCPoint1[3990] = {X 156.7436, Y 43.6961, Z -1.3333, A 0.000, B 0.000, C 0.000 }
gfCNCPoint1[3991] = {X 156.7578, Y 43.9498, Z -1.3333, A 0.000, B 0.000, C 0.000 }
gfCNCPoint1[3992] = {X 156.7631, Y 44.2039, Z -1.3333, A 0.000, B 0.000, C 0.000 }
gfCNCPoint1[3993] = {X 156.7629, Y 45.0588, Z -1.3333, A 0.000, B 0.000, C 0.000 }
gfCNCPoint1[3994] = {X 156.7352, Y 45.6370, Z -1.3333, A 0.000, B 0.000, C 0.000 }
gfCNCPoint1[3995] = {X 156.6616, Y 46.2112, Z -1.3333, A 0.000, B 0.000, C 0.000 }
gfCNCPoint1[3996] = {X 157.9051, Y 46.0006, Z -1.3333, A 0.000, B 0.000, C 0.000 }
gfCNCPoint1[3997] = {X 159.1638, Y 45.9207, Z -1.3333, A 0.000, B 0.000, C 0.000 }
gfCNCPoint1[3998] = {X 159.2309, Y 45.9202, Z -1.3333, A 0.000, B 0.000, C 0.000 }
gfCNCPoint1[3999] = {X 159.2980, Y 45.9200, Z -1.3333, A 0.000, B 0.000, C 0.000 }
gfCNCPoint1[4000] = {X 169.6843, Y 45.9200, Z -1.3333, A 0.000, B 0.000, C 0.000 }
gfCNCPoint1[4001] = {X 168.9035, Y 44.8481, Z -1.3333, A 0.000, B 0.000, C 0.000 }
gfCNCPoint1[4002] = {X 168.2131, Y 43.7159, Z -1.3333, A 0.000, B 0.000, C 0.000 }
gfCNCPoint1[4003] = {X 167.6176, Y 42.5310, Z -1.3333, A 0.000, B 0.000, C 0.000 }
gfCNCPoint1[4004] = {X 166.9496, Y 40.7947, Z -1.3333, A 0.000, B 0.000, C 0.000 }
gfCNCPoint1[4005] = {X 166.4851, Y 38.9932, Z -1.3333, A 0.000, B 0.000, C 0.000 }
gfCNCPoint1[4006] = {X 166.2304, Y 37.1503, Z -1.3333, A 0.000, B 0.000, C 0.000 }
gfCNCPoint1[4007] = {X 166.1319, Y 35.3980, Z -1.3333, A 0.000, B 0.000, C 0.000 }
gfCNCPoint1[4008] = {X 166.2084, Y 33.6446, Z -1.3333, A 0.000, B 0.000, C 0.000 }
gfCNCPoint1[4009] = {X 166.4594, Y 31.9075, Z -1.3333, A 0.000, B 0.000, C 0.000 }
gfCNCPoint1[4010] = {X 166.8822, Y 30.2041, Z -1.3333, A 0.000, B 0.000, C 0.000 }
gfCNCPoint1[4011] = {X 167.4726, Y 28.5514, Z -1.3333, A 0.000, B 0.000, C 0.000 }
gfCNCPoint1[4012] = {X 168.2336, Y 26.9822, Z -1.3333, A 0.000, B 0.000, C 0.000 }
gfCNCPoint1[4013] = {X 169.1861, Y 25.5212, Z -1.3333, A 0.000, B 0.000, C 0.000 }
gfCNCPoint1[4014] = {X 170.3149, Y 24.1918, Z -1.3333, A 0.000, B 0.000, C 0.000 }
gfCNCPoint1[4015] = {X 169.9867, Y 23.6227, Z -1.3333, A 0.000, B 0.000, C 0.000 }
gfCNCPoint1[4016] = {X 169.7113, Y 23.0264, Z -1.3333, A 0.000, B 0.000, C 0.000 }
gfCNCPoint1[4017] = {X 167.1001, Y 16.6309, Z -1.3333, A 0.000, B 0.000, C 0.000 }
gfCNCPoint1[4018] = {X 166.7820, Y 15.6636, Z -1.3333, A 0.000, B 0.000, C 0.000 }
gfCNCPoint1[4019] = {X 166.6021, Y 14.6613, Z -1.3333, A 0.000, B 0.000, C 0.000 }
gfCNCPoint1[4020] = {X 166.6021, Y 17.4615, Z -1.3333, A 0.000, B 0.000, C 0.000 }
gfCNCPoint1[4021] = {X 166.5130, Y 18.5970, Z -1.3333, A 0.000, B 0.000, C 0.000 }
gfCNCPoint1[4022] = {X 166.2479, Y 19.7047, Z -1.3333, A 0.000, B 0.000, C 0.000 }
gfCNCPoint1[4023] = {X 165.8132, Y 20.7575, Z -1.3333, A 0.000, B 0.000, C 0.000 }
gfCNCPoint1[4024] = {X 165.2197, Y 21.7296, Z -1.3333, A 0.000, B 0.000, C 0.000 }
gfCNCPoint1[4025] = {X 164.3788, Y 22.6987, Z -1.3333, A 0.000, B 0.000, C 0.000 }
gfCNCPoint1[4026] = {X 163.3808, Y 23.5052, Z -1.3333, A 0.000, B 0.000, C 0.000 }
gfCNCPoint1[4027] = {X 162.2567, Y 24.1238, Z -1.3333, A 0.000, B 0.000, C 0.000 }
gfCNCPoint1[4028] = {X 161.0415, Y 24.5356, Z -1.3333, A 0.000, B 0.000, C 0.000 }
gfCNCPoint1[4029] = {X 160.4746, Y 22.2035, Z -1.3333, A 0.000, B 0.000, C 0.000 }
gfCNCPoint1[4030] = {X 159.9025, Y 22.3069, Z -1.3333, A 0.000, B 0.000, C 0.000 }
gfCNCPoint1[4031] = {X 159.3220, Y 22.3415, Z -1.3333, A 0.000, B 0.000, C 0.000 }
gfCNCPoint1[4032] = {X 158.6806, Y 22.3415, Z -1.3333, A 0.000, B 0.000, C 0.000 }
gfCNCPoint1[4033] = {X 157.8823, Y 22.2729, Z -1.3333, A 0.000, B 0.000, C 0.000 }
gfCNCPoint1[4034] = {X 157.1058, Y 22.0757, Z -1.3333, A 0.000, B 0.000, C 0.000 }
gfCNCPoint1[4035] = {X 156.3716, Y 21.7550, Z -1.3333, A 0.000, B 0.000, C 0.000 }
gfCNCPoint1[4036] = {X 155.5230, Y 21.1772, Z -1.3333, A 0.000, B 0.000, C 0.000 }
gfCNCPoint1[4037] = {X 154.8127, Y 20.4358, Z -1.3333, A 0.000, B 0.000, C 0.000 }
gfCNCPoint1[4038] = {X 152.8355, Y 20.4368, Z -1.3333, A 0.000, B 0.000, C 0.000 }
gfCNCPoint1[4039] = {X 152.8338, Y 40.6542, Z -1.3333, A 0.000, B 0.000, C 0.000 }
gfCNCPoint1[4040] = {X 153.1758, Y 41.0241, Z -1.3333, A 0.000, B 0.000, C 0.000 }
gfCNCPoint1[4041] = {X 153.6800, Y 41.7287, Z -1.3333, A 0.000, B 0.000, C 0.000 }
gfCNCPoint1[4042] = {X 154.0530, Y 42.5108, Z -1.3333, A 0.000, B 0.000, C 0.000 }
gfCNCPoint1[4043] = {X 154.2830, Y 43.3462, Z -1.3333, A 0.000, B 0.000, C 0.000 }
gfCNCPoint1[4044] = {X 154.3631, Y 44.2089, Z -1.3333, A 0.000, B 0.000, C 0.000 }
gfCNCPoint1[4045] = {X 154.3629, Y 45.0469, Z -1.3333, A 0.000, B 0.000, C 0.000 }
gfCNCPoint1[4046] = {X 154.3440, Y 45.4308, Z -1.3333, A 0.000, B 0.000, C 0.000 }
gfCNCPoint1[4047] = {X 154.2951, Y 45.8119, Z -1.3333, A 0.000, B 0.000, C 0.000 }
gfCNCPoint1[4048] = {X 154.0370, Y 46.7541, Z -1.3333, A 0.000, B 0.000, C 0.000 }
gfCNCPoint1[4049] = {X 153.5963, Y 47.6260, Z -1.3333, A 0.000, B 0.000, C 0.000 }
gfCNCPoint1[4050] = {X 152.9909, Y 48.3926, Z -1.3333, A 0.000, B 0.000, C 0.000 }
gfCNCPoint1[4051] = {X 152.2448, Y 49.0233, Z -1.3333, A 0.000, B 0.000, C 0.000 }
gfCNCPoint1[4052] = {X 151.3881, Y 49.4928, Z -1.3333, A 0.000, B 0.000, C 0.000 }
gfCNCPoint1[4053] = {X 150.4551, Y 49.7822, Z -1.3333, A 0.000, B 0.000, C 0.000 }
gfCNCPoint1[4054] = {X 149.4831, Y 49.8800, Z -1.3333, A 0.000, B 0.000, C 0.000 }
gfCNCPoint1[4055] = {X 143.0396, Y 49.8800, Z -1.3333, A 0.000, B 0.000, C 0.000 }
gfCNCPoint1[4056] = {X 142.0923, Y 49.7872, Z -1.3333, A 0.000, B 0.000, C 0.000 }
gfCNCPoint1[4057] = {X 141.1811, Y 49.5122, Z -1.3333, A 0.000, B 0.000, C 0.000 }
gfCNCPoint1[4058] = {X 140.3405, Y 49.0656, Z -1.3333, A 0.000, B 0.000, C 0.000 }
gfCNCPoint1[4059] = {X 139.6026, Y 48.4643, Z -1.3333, A 0.000, B 0.000, C 0.000 }
gfCNCPoint1[4060] = {X 138.9955, Y 47.7312, Z -1.3333, A 0.000, B 0.000, C 0.000 }
gfCNCPoint1[4061] = {X 138.5423, Y 46.8942, Z -1.3333, A 0.000, B 0.000, C 0.000 }
gfCNCPoint1[4062] = {X 138.2601, Y 45.9852, Z -1.3333, A 0.000, B 0.000, C 0.000 }
gfCNCPoint1[4063] = {X 138.1598, Y 45.0386, Z -1.3333, A 0.000, B 0.000, C 0.000 }
gfCNCPoint1[4064] = {X 138.1601, Y 44.1416, Z -1.3333, A 0.000, B 0.000, C 0.000 }
gfCNCPoint1[4065] = {X 138.2148, Y 43.4769, Z -1.3333, A 0.000, B 0.000, C 0.000 }
gfCNCPoint1[4066] = {X 138.3597, Y 42.8258, Z -1.3333, A 0.000, B 0.000, C 0.000 }
gfCNCPoint1[4067] = {X 129.1532, Y 40.1052, Z -1.3333, A 0.000, B 0.000, C 0.000 }
gfCNCPoint1[4068] = {X 129.5665, Y 38.9035, Z -1.3333, A 0.000, B 0.000, C 0.000 }
gfCNCPoint1[4069] = {X 130.0836, Y 37.7426, Z -1.3333, A 0.000, B 0.000, C 0.000 }
gfCNCPoint1[4070] = {X 130.0836, Y 31.6021, Z -1.3333, A 0.000, B 0.000, C 0.000 }
gfCNCPoint1[4071] = {X 129.2057, Y 31.3795, Z -1.3333, A 0.000, B 0.000, C 0.000 }
gfCNCPoint1[4072] = {X 128.3433, Y 31.1025, Z -1.3333, A 0.000, B 0.000, C 0.000 }
gfCNCPoint1[4073] = {X 128.3430, Y 38.3271, Z -1.3333, A 0.000, B 0.000, C 0.000 }
gfCNCPoint1[4074] = {X 128.7841, Y 39.1998, Z -1.3333, A 0.000, B 0.000, C 0.000 }
gfCNCPoint1[4075] = {X 129.1532, Y 40.1052, Z -1.3333, A 0.000, B 0.000, C 0.000 }
gfCNCPoint1[4076] = {X 131.4548, Y 40.7854, Z -1.3333, A 0.000, B 0.000, C 0.000 }
gfCNCPoint1[4077] = {X 131.9017, Y 39.5320, Z -1.3333, A 0.000, B 0.000, C 0.000 }
gfCNCPoint1[4078] = {X 132.4836, Y 38.3354, Z -1.3333, A 0.000, B 0.000, C 0.000 }
gfCNCPoint1[4079] = {X 132.4836, Y 29.5202, Z -1.3333, A 0.000, B 0.000, C 0.000 }
gfCNCPoint1[4080] = {X 131.3522, Y 29.3993, Z -1.3333, A 0.000, B 0.000, C 0.000 }
gfCNCPoint1[4081] = {X 130.2371, Y 29.1724, Z -1.3333, A 0.000, B 0.000, C 0.000 }
gfCNCPoint1[4082] = {X 129.1484, Y 28.8416, Z -1.3333, A 0.000, B 0.000, C 0.000 }
gfCNCPoint1[4083] = {X 128.0240, Y 28.3761, Z -1.3333, A 0.000, B 0.000, C 0.000 }
gfCNCPoint1[4084] = {X 126.9520, Y 27.7999, Z -1.3333, A 0.000, B 0.000, C 0.000 }
gfCNCPoint1[4085] = {X 125.9435, Y 27.1187, Z -1.3333, A 0.000, B 0.000, C 0.000 }
gfCNCPoint1[4086] = {X 125.9429, Y 38.9879, Z -1.3333, A 0.000, B 0.000, C 0.000 }
gfCNCPoint1[4087] = {X 126.4734, Y 39.9276, Z -1.3333, A 0.000, B 0.000, C 0.000 }
gfCNCPoint1[4088] = {X 126.8960, Y 40.9205, Z -1.3333, A 0.000, B 0.000, C 0.000 }
gfCNCPoint1[4089] = {X 127.2098, Y 41.9730, Z -1.3333, A 0.000, B 0.000, C 0.000 }
gfCNCPoint1[4090] = {X 127.4025, Y 43.0542, Z -1.3333, A 0.000, B 0.000, C 0.000 }
gfCNCPoint1[4091] = {X 127.4714, Y 44.1502, Z -1.3333, A 0.000, B 0.000, C 0.000 }
gfCNCPoint1[4092] = {X 127.4716, Y 45.0000, Z -1.3333, A 0.000, B 0.000, C 0.000 }
gfCNCPoint1[4093] = {X 127.4070, Y 46.1159, Z -1.3333, A 0.000, B 0.000, C 0.000 }
gfCNCPoint1[4094] = {X 127.2143, Y 47.2168, Z -1.3333, A 0.000, B 0.000, C 0.000 }
gfCNCPoint1[4095] = {X 126.8960, Y 48.2883, Z -1.3333, A 0.000, B 0.000, C 0.000 }
gfCNCPoint1[4096] = {X 126.2883, Y 49.6376, Z -1.3333, A 0.000, B 0.000, C 0.000 }
gfCNCPoint1[4097] = {X 125.4821, Y 50.8786, Z -1.3333, A 0.000, B 0.000, C 0.000 }
gfCNCPoint1[4098] = {X 124.4962, Y 51.9821, Z -1.3333, A 0.000, B 0.000, C 0.000 }
gfCNCPoint1[4099] = {X 123.3536, Y 52.9225, Z -1.3333, A 0.000, B 0.000, C 0.000 }
gfCNCPoint1[4100] = {X 122.0810, Y 53.6778, Z -1.3333, A 0.000, B 0.000, C 0.000 }
gfCNCPoint1[4101] = {X 120.7081, Y 54.2302, Z -1.3333, A 0.000, B 0.000, C 0.000 }
gfCNCPoint1[4102] = {X 119.2671, Y 54.5669, Z -1.3333, A 0.000, B 0.000, C 0.000 }
gfCNCPoint1[4103] = {X 117.7916, Y 54.6800, Z -1.3333, A 0.000, B 0.000, C 0.000 }
gfCNCPoint1[4104] = {X 111.9185, Y 54.6800, Z -1.3333, A 0.000, B 0.000, C 0.000 }
gfCNCPoint1[4105] = {X 111.7456, Y 54.6785, Z -1.3333, A 0.000, B 0.000, C 0.000 }
gfCNCPoint1[4106] = {X 111.5728, Y 54.6738, Z -1.3333, A 0.000, B 0.000, C 0.000 }
gfCNCPoint1[4107] = {X 111.0585, Y 69.0646, Z -1.3333, A 0.000, B 0.000, C 0.000 }
gfCNCPoint1[4108] = {X 109.0296, Y 68.9061, Z -1.3333, A 0.000, B 0.000, C 0.000 }
gfCNCPoint1[4109] = {X 107.0213, Y 68.5768, Z -1.3333, A 0.000, B 0.000, C 0.000 }
gfCNCPoint1[4110] = {X 105.0765, Y 68.8983, Z -1.3333, A 0.000, B 0.000, C 0.000 }
gfCNCPoint1[4111] = {X 103.1119, Y 69.0597, Z -1.3333, A 0.000, B 0.000, C 0.000 }
gfCNCPoint1[4112] = {X 101.1407, Y 69.0599, Z -1.3333, A 0.000, B 0.000, C 0.000 }
gfCNCPoint1[4113] = {X 99.1761, Y 68.8989, Z -1.3333, A 0.000, B 0.000, C 0.000 }
gfCNCPoint1[4114] = {X 97.2313, Y 68.5777, Z -1.3333, A 0.000, B 0.000, C 0.000 }
gfCNCPoint1[4115] = {X 95.6131, Y 68.8563, Z -1.3333, A 0.000, B 0.000, C 0.000 }
gfCNCPoint1[4116] = {X 93.9796, Y 69.0240, Z -1.3333, A 0.000, B 0.000, C 0.000 }
gfCNCPoint1[4117] = {X 92.3385, Y 69.0800, Z -1.3333, A 0.000, B 0.000, C 0.000 }
gfCNCPoint1[4118] = {X 86.6884, Y 69.0800, Z -1.3333, A 0.000, B 0.000, C 0.000 }
gfCNCPoint1[4119] = {X 84.7318, Y 70.2668, Z -1.3333, A 0.000, B 0.000, C 0.000 }
gfCNCPoint1[4120] = {X 82.6874, Y 71.2949, Z -1.3333, A 0.000, B 0.000, C 0.000 }
gfCNCPoint1[4121] = {X 107.2717, Y 71.2949, Z -1.3333, A 0.000, B 0.000, C 0.000 }
gfCNCPoint1[4122] = {X 109.1259, Y 70.1132, Z -1.3333, A 0.000, B 0.000, C 0.000 }
gfCNCPoint1[4123] = {X 111.0585, Y 69.0646, Z -1.3333, A 0.000, B 0.000, C 0.000 }
gfCNCPoint1[4124] = {X 111.1442, Y 66.6662, Z -1.3333, A 0.000, B 0.000, C 0.000 }
gfCNCPoint1[4125] = {X 109.0696, Y 66.4920, Z -1.3333, A 0.000, B 0.000, C 0.000 }
gfCNCPoint1[4126] = {X 107.0213, Y 66.1197, Z -1.3333, A 0.000, B 0.000, C 0.000 }
gfCNCPoint1[4127] = {X 105.0796, Y 66.4776, Z -1.3333, A 0.000, B 0.000, C 0.000 }
gfCNCPoint1[4128] = {X 103.1135, Y 66.6574, Z -1.3333, A 0.000, B 0.000, C 0.000 }
gfCNCPoint1[4129] = {X 101.1392, Y 66.6576, Z -1.3333, A 0.000, B 0.000, C 0.000 }
gfCNCPoint1[4130] = {X 99.1730, Y 66.4782, Z -1.3333, A 0.000, B 0.000, C 0.000 }
gfCNCPoint1[4131] = {X 97.2313, Y 66.1207, Z -1.3333, A 0.000, B 0.000, C 0.000 }
gfCNCPoint1[4132] = {X 95.6161, Y 66.4308, Z -1.3333, A 0.000, B 0.000, C 0.000 }
gfCNCPoint1[4133] = {X 93.9821, Y 66.6176, Z -1.3333, A 0.000, B 0.000, C 0.000 }
gfCNCPoint1[4134] = {X 92.3385, Y 66.6800, Z -1.3333, A 0.000, B 0.000, C 0.000 }
gfCNCPoint1[4135] = {X 85.9487, Y 66.6800, Z -1.3333, A 0.000, B 0.000, C 0.000 }
gfCNCPoint1[4136] = {X 83.8781, Y 67.9934, Z -1.3333, A 0.000, B 0.000, C 0.000 }
gfCNCPoint1[4137] = {X 81.6949, Y 69.1097, Z -1.3333, A 0.000, B 0.000, C 0.000 }
gfCNCPoint1[4138] = {X 79.6018, Y 69.9547, Z -1.3333, A 0.000, B 0.000, C 0.000 }
gfCNCPoint1[4139] = {X 77.4444, Y 70.6184, Z -1.3333, A 0.000, B 0.000, C 0.000 }
gfCNCPoint1[4140] = {X 75.2383, Y 71.0959, Z -1.3333, A 0.000, B 0.000, C 0.000 }
gfCNCPoint1[4141] = {X 72.9996, Y 71.3838, Z -1.3333, A 0.000, B 0.000, C 0.000 }
gfCNCPoint1[4142] = {X 70.7445, Y 71.4800, Z -1.3333, A 0.000, B 0.000, C 0.000 }
gfCNCPoint1[4143] = {X 64.1851, Y 71.4800, Z -1.3333, A 0.000, B 0.000, C 0.000 }
gfCNCPoint1[4144] = {X 62.0752, Y 71.3958, Z -1.3333, A 0.000, B 0.000, C 0.000 }
gfCNCPoint1[4145] = {X 59.9787, Y 71.1438, Z -1.3333, A 0.000, B 0.000, C 0.000 }
gfCNCPoint1[4146] = {X 57.9089, Y 70.7255, Z -1.3333, A 0.000, B 0.000, C 0.000 }
gfCNCPoint1[4147] = {X 55.8790, Y 70.1436, Z -1.3333, A 0.000, B 0.000, C 0.000 }
gfCNCPoint1[4148] = {X 53.8492, Y 70.7255, Z -1.3333, A 0.000, B 0.000, C 0.000 }
gfCNCPoint1[4149] = {X 51.7794, Y 71.1438, Z -1.3333, A 0.000, B 0.000, C 0.000 }
gfCNCPoint1[4150] = {X 49.6829, Y 71.3958, Z -1.3333, A 0.000, B 0.000, C 0.000 }
gfCNCPoint1[4151] = {X 47.5729, Y 71.4800, Z -1.3333, A 0.000, B 0.000, C 0.000 }
gfCNCPoint1[4152] = {X 40.6393, Y 71.4800, Z -1.3333, A 0.000, B 0.000, C 0.000 }
gfCNCPoint1[4153] = {X 38.8039, Y 71.4163, Z -1.3333, A 0.000, B 0.000, C 0.000 }
gfCNCPoint1[4154] = {X 36.9773, Y 71.2256, Z -1.3333, A 0.000, B 0.000, C 0.000 }
gfCNCPoint1[4155] = {X 34.3995, Y 72.0336, Z -1.3333, A 0.000, B 0.000, C 0.000 }
gfCNCPoint1[4156] = {X 31.7608, Y 72.6128, Z -1.3333, A 0.000, B 0.000, C 0.000 }
gfCNCPoint1[4157] = {X 30.3286, Y 73.1740, Z -1.3333, A 0.000, B 0.000, C 0.000 }
gfCNCPoint1[4158] = {X 28.8811, Y 73.6949, Z -1.3333, A 0.000, B 0.000, C 0.000 }
gfCNCPoint1[4159] = {X 108.0339, Y 73.6949, Z -1.3333, A 0.000, B 0.000, C 0.000 }
gfCNCPoint1[4160] = {X 110.0295, Y 72.3690, Z -1.3333, A 0.000, B 0.000, C 0.000 }
gfCNCPoint1[4161] = {X 112.1282, Y 71.2131, Z -1.3333, A 0.000, B 0.000, C 0.000 }
gfCNCPoint1[4162] = {X 113.1276, Y 70.7391, Z -1.3333, A 0.000, B 0.000, C 0.000 }
gfCNCPoint1[4163] = {X 114.1445, Y 70.3038, Z -1.3333, A 0.000, B 0.000, C 0.000 }
gfCNCPoint1[4164] = {X 117.4444, Y 66.6800, Z -1.3333, A 0.000, B 0.000, C 0.000 }
gfCNCPoint1[4165] = {X 111.9185, Y 66.6800, Z -1.3333, A 0.000, B 0.000, C 0.000 }
gfCNCPoint1[4166] = {X 111.5313, Y 66.6765, Z -1.3333, A 0.000, B 0.000, C 0.000 }
gfCNCPoint1[4167] = {X 111.1442, Y 66.6662, Z -1.3333, A 0.000, B 0.000, C 0.000 }
gfCNCPoint1[4168] = {X 111.2299, Y 64.2677, Z -1.3333, A 0.000, B 0.000, C 0.000 }
gfCNCPoint1[4169] = {X 109.1084, Y 64.0741, Z -1.3333, A 0.000, B 0.000, C 0.000 }
gfCNCPoint1[4170] = {X 107.0213, Y 63.6477, Z -1.3333, A 0.000, B 0.000, C 0.000 }
gfCNCPoint1[4171] = {X 105.0841, Y 64.0514, Z -1.3333, A 0.000, B 0.000, C 0.000 }
gfCNCPoint1[4172] = {X 103.1158, Y 64.2545, Z -1.3333, A 0.000, B 0.000, C 0.000 }
gfCNCPoint1[4173] = {X 101.1370, Y 64.2547, Z -1.3333, A 0.000, B 0.000, C 0.000 }
gfCNCPoint1[4174] = {X 99.1686, Y 64.0521, Z -1.3333, A 0.000, B 0.000, C 0.000 }
gfCNCPoint1[4175] = {X 97.2313, Y 63.6488, Z -1.3333, A 0.000, B 0.000, C 0.000 }
gfCNCPoint1[4176] = {X 95.6204, Y 63.9986, Z -1.3333, A 0.000, B 0.000, C 0.000 }
gfCNCPoint1[4177] = {X 93.9855, Y 64.2095, Z -1.3333, A 0.000, B 0.000, C 0.000 }
gfCNCPoint1[4178] = {X 92.3385, Y 64.2800, Z -1.3333, A 0.000, B 0.000, C 0.000 }
gfCNCPoint1[4179] = {X 85.8951, Y 64.2800, Z -1.3333, A 0.000, B 0.000, C 0.000 }
gfCNCPoint1[4180] = {X 85.5417, Y 64.2768, Z -1.3333, A 0.000, B 0.000, C 0.000 }
gfCNCPoint1[4181] = {X 85.1884, Y 64.2670, Z -1.3333, A 0.000, B 0.000, C 0.000 }
gfCNCPoint1[4182] = {X 83.3593, Y 65.5113, Z -1.3333, A 0.000, B 0.000, C 0.000 }
gfCNCPoint1[4183] = {X 81.4238, Y 66.5824, Z -1.3333, A 0.000, B 0.000, C 0.000 }
gfCNCPoint1[4184] = {X 79.3981, Y 67.4713, Z -1.3333, A 0.000, B 0.000, C 0.000 }
gfCNCPoint1[4185] = {X 77.2994, Y 68.1706, Z -1.3333, A 0.000, B 0.000, C 0.000 }
gfCNCPoint1[4186] = {X 75.1454, Y 68.6744, Z -1.3333, A 0.000, B 0.000, C 0.000 }
gfCNCPoint1[4187] = {X 72.9543, Y 68.9784, Z -1.3333, A 0.000, B 0.000, C 0.000 }
gfCNCPoint1[4188] = {X 70.7445, Y 69.0800, Z -1.3333, A 0.000, B 0.000, C 0.000 }
gfCNCPoint1[4189] = {X 64.1851, Y 69.0800, Z -1.3333, A 0.000, B 0.000, C 0.000 }
gfCNCPoint1[4190] = {X 62.0678, Y 68.9867, Z -1.3333, A 0.000, B 0.000, C 0.000 }
gfCNCPoint1[4191] = {X 59.9669, Y 68.7076, Z -1.3333, A 0.000, B 0.000, C 0.000 }
gfCNCPoint1[4192] = {X 57.8986, Y 68.2449, Z -1.3333, A 0.000, B 0.000, C 0.000 }
gfCNCPoint1[4193] = {X 55.8790, Y 67.6021, Z -1.3333, A 0.000, B 0.000, C 0.000 }
gfCNCPoint1[4194] = {X 53.8595, Y 68.2449, Z -1.3333, A 0.000, B 0.000, C 0.000 }
gfCNCPoint1[4195] = {X 51.7912, Y 68.7076, Z -1.3333, A 0.000, B 0.000, C 0.000 }
gfCNCPoint1[4196] = {X 49.6903, Y 68.9867, Z -1.3333, A 0.000, B 0.000, C 0.000 }
gfCNCPoint1[4197] = {X 47.5729, Y 69.0800, Z -1.3333, A 0.000, B 0.000, C 0.000 }
gfCNCPoint1[4198] = {X 40.6393, Y 69.0800, Z -1.3333, A 0.000, B 0.000, C 0.000 }
gfCNCPoint1[4199] = {X 38.6735, Y 68.9996, Z -1.3333, A 0.000, B 0.000, C 0.000 }
gfCNCPoint1[4200] = {X 36.7209, Y 68.7591, Z -1.3333, A 0.000, B 0.000, C 0.000 }
gfCNCPoint1[4201] = {X 34.8825, Y 69.3979, Z -1.3333, A 0.000, B 0.000, C 0.000 }
gfCNCPoint1[4202] = {X 33.0046, Y 69.9094, Z -1.3333, A 0.000, B 0.000, C 0.000 }
gfCNCPoint1[4203] = {X 31.0961, Y 70.2912, Z -1.3333, A 0.000, B 0.000, C 0.000 }
gfCNCPoint1[4204] = {X 29.6068, Y 70.8812, Z -1.3333, A 0.000, B 0.000, C 0.000 }
gfCNCPoint1[4205] = {X 28.1002, Y 71.4255, Z -1.3333, A 0.000, B 0.000, C 0.000 }
gfCNCPoint1[4206] = {X 26.8254, Y 71.8460, Z -1.3333, A 0.000, B 0.000, C 0.000 }
gfCNCPoint1[4207] = {X 25.5403, Y 72.2338, Z -1.3333, A 0.000, B 0.000, C 0.000 }
gfCNCPoint1[4208] = {X 24.8758, Y 72.4184, Z -1.3333, A 0.000, B 0.000, C 0.000 }
gfCNCPoint1[4209] = {X 24.3904, Y 72.5501, Z -1.3333, A 0.000, B 0.000, C 0.000 }
gfCNCPoint1[4210] = {X 23.9035, Y 72.6765, Z -1.3333, A 0.000, B 0.000, C 0.000 }
gfCNCPoint1[4211] = {X 23.9035, Y 76.0949, Z -1.3333, A 0.000, B 0.000, C 0.000 }
gfCNCPoint1[4212] = {X 108.8320, Y 76.0949, Z -1.3333, A 0.000, B 0.000, C 0.000 }
gfCNCPoint1[4213] = {X 110.4024, Y 74.9730, Z -1.3333, A 0.000, B 0.000, C 0.000 }
gfCNCPoint1[4214] = {X 112.0503, Y 73.9684, Z -1.3333, A 0.000, B 0.000, C 0.000 }
gfCNCPoint1[4215] = {X 113.7671, Y 73.0865, Z -1.3333, A 0.000, B 0.000, C 0.000 }
gfCNCPoint1[4216] = {X 115.5435, Y 72.3321, Z -1.3333, A 0.000, B 0.000, C 0.000 }
gfCNCPoint1[4217] = {X 123.7293, Y 63.3429, Z -1.3333, A 0.000, B 0.000, C 0.000 }
gfCNCPoint1[4218] = {X 121.7863, Y 63.8616, Z -1.3333, A 0.000, B 0.000, C 0.000 }
gfCNCPoint1[4219] = {X 119.7999, Y 64.1751, Z -1.3333, A 0.000, B 0.000, C 0.000 }
gfCNCPoint1[4220] = {X 117.7916, Y 64.2800, Z -1.3333, A 0.000, B 0.000, C 0.000 }
gfCNCPoint1[4221] = {X 111.9185, Y 64.2800, Z -1.3333, A 0.000, B 0.000, C 0.000 }
gfCNCPoint1[4222] = {X 111.5741, Y 64.2769, Z -1.3333, A 0.000, B 0.000, C 0.000 }
gfCNCPoint1[4223] = {X 111.2299, Y 64.2677, Z -1.3333, A 0.000, B 0.000, C 0.000 }
gfCNCPoint1[4224] = {X 111.3156, Y 61.8692, Z -1.3333, A 0.000, B 0.000, C 0.000 }
gfCNCPoint1[4225] = {X 109.8654, Y 61.7547, Z -1.3333, A 0.000, B 0.000, C 0.000 }
gfCNCPoint1[4226] = {X 108.4304, Y 61.5157, Z -1.3333, A 0.000, B 0.000, C 0.000 }
gfCNCPoint1[4227] = {X 107.0213, Y 61.1540, Z -1.3333, A 0.000, B 0.000, C 0.000 }
gfCNCPoint1[4228] = {X 105.0907, Y 61.6173, Z -1.3333, A 0.000, B 0.000, C 0.000 }
gfCNCPoint1[4229] = {X 103.1191, Y 61.8506, Z -1.3333, A 0.000, B 0.000, C 0.000 }
gfCNCPoint1[4230] = {X 101.1337, Y 61.8509, Z -1.3333, A 0.000, B 0.000, C 0.000 }
gfCNCPoint1[4231] = {X 99.1620, Y 61.6181, Z -1.3333, A 0.000, B 0.000, C 0.000 }
gfCNCPoint1[4232] = {X 97.2313, Y 61.1553, Z -1.3333, A 0.000, B 0.000, C 0.000 }
gfCNCPoint1[4233] = {X 95.6267, Y 61.5566, Z -1.3333, A 0.000, B 0.000, C 0.000 }
gfCNCPoint1[4234] = {X 93.9906, Y 61.7990, Z -1.3333, A 0.000, B 0.000, C 0.000 }
gfCNCPoint1[4235] = {X 92.3385, Y 61.8800, Z -1.3333, A 0.000, B 0.000, C 0.000 }
gfCNCPoint1[4236] = {X 85.8951, Y 61.8800, Z -1.3333, A 0.000, B 0.000, C 0.000 }
gfCNCPoint1[4237] = {X 85.1609, Y 61.8640, Z -1.3333, A 0.000, B 0.000, C 0.000 }
gfCNCPoint1[4238] = {X 84.4280, Y 61.8161, Z -1.3333, A 0.000, B 0.000, C 0.000 }
gfCNCPoint1[4239] = {X 82.7247, Y 63.0692, Z -1.3333, A 0.000, B 0.000, C 0.000 }
gfCNCPoint1[4240] = {X 80.9073, Y 64.1504, Z -1.3333, A 0.000, B 0.000, C 0.000 }
gfCNCPoint1[4241] = {X 78.9932, Y 65.0494, Z -1.3333, A 0.000, B 0.000, C 0.000 }
gfCNCPoint1[4242] = {X 77.0007, Y 65.7577, Z -1.3333, A 0.000, B 0.000, C 0.000 }
gfCNCPoint1[4243] = {X 74.9487, Y 66.2685, Z -1.3333, A 0.000, B 0.000, C 0.000 }
gfCNCPoint1[4244] = {X 72.8566, Y 66.5769, Z -1.3333, A 0.000, B 0.000, C 0.000 }
gfCNCPoint1[4245] = {X 70.7445, Y 66.6800, Z -1.3333, A 0.000, B 0.000, C 0.000 }
gfCNCPoint1[4246] = {X 64.1851, Y 66.6800, Z -1.3333, A 0.000, B 0.000, C 0.000 }
gfCNCPoint1[4247] = {X 62.0576, Y 66.5754, Z -1.3333, A 0.000, B 0.000, C 0.000 }
gfCNCPoint1[4248] = {X 59.9505, Y 66.2624, Z -1.3333, A 0.000, B 0.000, C 0.000 }
gfCNCPoint1[4249] = {X 57.8844, Y 65.7442, Z -1.3333, A 0.000, B 0.000, C 0.000 }
gfCNCPoint1[4250] = {X 55.8790, Y 65.0258, Z -1.3333, A 0.000, B 0.000, C 0.000 }
gfCNCPoint1[4251] = {X 53.8737, Y 65.7442, Z -1.3333, A 0.000, B 0.000, C 0.000 }
gfCNCPoint1[4252] = {X 51.8075, Y 66.2624, Z -1.3333, A 0.000, B 0.000, C 0.000 }
gfCNCPoint1[4253] = {X 49.7005, Y 66.5754, Z -1.3333, A 0.000, B 0.000, C 0.000 }
gfCNCPoint1[4254] = {X 47.5729, Y 66.6800, Z -1.3333, A 0.000, B 0.000, C 0.000 }
gfCNCPoint1[4255] = {X 40.6393, Y 66.6800, Z -1.3333, A 0.000, B 0.000, C 0.000 }
gfCNCPoint1[4256] = {X 38.5438, Y 66.5785, Z -1.3333, A 0.000, B 0.000, C 0.000 }
gfCNCPoint1[4257] = {X 36.4680, Y 66.2749, Z -1.3333, A 0.000, B 0.000, C 0.000 }
gfCNCPoint1[4258] = {X 34.5049, Y 67.0000, Z -1.3333, A 0.000, B 0.000, C 0.000 }
gfCNCPoint1[4259] = {X 32.4899, Y 67.5650, Z -1.3333, A 0.000, B 0.000, C 0.000 }
gfCNCPoint1[4260] = {X 30.4360, Y 67.9662, Z -1.3333, A 0.000, B 0.000, C 0.000 }
gfCNCPoint1[4261] = {X 27.6849, Y 69.0287, Z -1.3333, A 0.000, B 0.000, C 0.000 }
gfCNCPoint1[4262] = {X 24.8761, Y 69.9276, Z -1.3333, A 0.000, B 0.000, C 0.000 }
gfCNCPoint1[4263] = {X 24.2350, Y 70.1056, Z -1.3333, A 0.000, B 0.000, C 0.000 }
gfCNCPoint1[4264] = {X 22.8746, Y 70.4592, Z -1.3333, A 0.000, B 0.000, C 0.000 }
gfCNCPoint1[4265] = {X 21.5035, Y 70.7691, Z -1.3333, A 0.000, B 0.000, C 0.000 }
gfCNCPoint1[4266] = {X 21.5035, Y 78.4949, Z -1.3333, A 0.000, B 0.000, C 0.000 }
gfCNCPoint1[4267] = {X 109.6715, Y 78.4949, Z -1.3333, A 0.000, B 0.000, C 0.000 }
gfCNCPoint1[4268] = {X 111.3433, Y 77.2331, Z -1.3333, A 0.000, B 0.000, C 0.000 }
gfCNCPoint1[4269] = {X 113.1183, Y 76.1214, Z -1.3333, A 0.000, B 0.000, C 0.000 }
gfCNCPoint1[4270] = {X 114.9833, Y 75.1682, Z -1.3333, A 0.000, B 0.000, C 0.000 }
gfCNCPoint1[4271] = {X 116.9240, Y 74.3806, Z -1.3333, A 0.000, B 0.000, C 0.000 }
gfCNCPoint1[4272] = {X 130.4119, Y 59.5691, Z -1.3333, A 0.000, B 0.000, C 0.000 }
gfCNCPoint1[4273] = {X 129.5281, Y 58.7535, Z -1.3333, A 0.000, B 0.000, C 0.000 }
gfCNCPoint1[4274] = {X 128.6970, Y 57.8844, Z -1.3333, A 0.000, B 0.000, C 0.000 }
gfCNCPoint1[4275] = {X 127.3932, Y 58.8832, Z -1.3333, A 0.000, B 0.000, C 0.000 }
gfCNCPoint1[4276] = {X 125.9986, Y 59.7506, Z -1.3333, A 0.000, B 0.000, C 0.000 }
gfCNCPoint1[4277] = {X 124.5262, Y 60.4783, Z -1.3333, A 0.000, B 0.000, C 0.000 }
gfCNCPoint1[4278] = {X 122.9902, Y 61.0595, Z -1.3333, A 0.000, B 0.000, C 0.000 }
gfCNCPoint1[4279] = {X 121.2890, Y 61.5137, Z -1.3333, A 0.000, B 0.000, C 0.000 }
gfCNCPoint1[4280] = {X 119.5499, Y 61.7882, Z -1.3333, A 0.000, B 0.000, C 0.000 }
gfCNCPoint1[4281] = {X 117.7916, Y 61.8800, Z -1.3333, A 0.000, B 0.000, C 0.000 }
gfCNCPoint1[4282] = {X 111.9185, Y 61.8800, Z -1.3333, A 0.000, B 0.000, C 0.000 }
gfCNCPoint1[4283] = {X 111.6170, Y 61.8773, Z -1.3333, A 0.000, B 0.000, C 0.000 }
gfCNCPoint1[4284] = {X 111.3156, Y 61.8692, Z -1.3333, A 0.000, B 0.000, C 0.000 }
gfCNCPoint1[4285] = {X 111.4013, Y 59.4708, Z -1.3333, A 0.000, B 0.000, C 0.000 }
gfCNCPoint1[4286] = {X 109.9149, Y 59.3407, Z -1.3333, A 0.000, B 0.000, C 0.000 }
gfCNCPoint1[4287] = {X 108.4496, Y 59.0584, Z -1.3333, A 0.000, B 0.000, C 0.000 }
gfCNCPoint1[4288] = {X 107.0213, Y 58.6267, Z -1.3333, A 0.000, B 0.000, C 0.000 }
gfCNCPoint1[4289] = {X 105.4260, Y 59.0985, Z -1.3333, A 0.000, B 0.000, C 0.000 }
gfCNCPoint1[4290] = {X 103.7872, Y 59.3842, Z -1.3333, A 0.000, B 0.000, C 0.000 }
gfCNCPoint1[4291] = {X 102.1264, Y 59.4800, Z -1.3333, A 0.000, B 0.000, C 0.000 }
gfCNCPoint1[4292] = {X 100.4656, Y 59.3847, Z -1.3333, A 0.000, B 0.000, C 0.000 }
gfCNCPoint1[4293] = {X 98.8267, Y 59.0996, Z -1.3333, A 0.000, B 0.000, C 0.000 }
gfCNCPoint1[4294] = {X 97.2313, Y 58.6283, Z -1.3333, A 0.000, B 0.000, C 0.000 }
gfCNCPoint1[4295] = {X 95.6367, Y 59.0994, Z -1.3333, A 0.000, B 0.000, C 0.000 }
gfCNCPoint1[4296] = {X 93.9986, Y 59.3845, Z -1.3333, A 0.000, B 0.000, C 0.000 }
gfCNCPoint1[4297] = {X 92.3385, Y 59.4800, Z -1.3333, A 0.000, B 0.000, C 0.000 }
gfCNCPoint1[4298] = {X 85.8951, Y 59.4800, Z -1.3333, A 0.000, B 0.000, C 0.000 }
gfCNCPoint1[4299] = {X 84.7780, Y 59.4368, Z -1.3333, A 0.000, B 0.000, C 0.000 }
gfCNCPoint1[4300] = {X 83.6677, Y 59.3077, Z -1.3333, A 0.000, B 0.000, C 0.000 }
gfCNCPoint1[4301] = {X 82.0978, Y 60.5827, Z -1.3333, A 0.000, B 0.000, C 0.000 }
gfCNCPoint1[4302] = {X 80.4031, Y 61.6862, Z -1.3333, A 0.000, B 0.000, C 0.000 }
gfCNCPoint1[4303] = {X 78.6021, Y 62.6061, Z -1.3333, A 0.000, B 0.000, C 0.000 }
gfCNCPoint1[4304] = {X 76.7146, Y 63.3324, Z -1.3333, A 0.000, B 0.000, C 0.000 }
gfCNCPoint1[4305] = {X 74.7614, Y 63.8569, Z -1.3333, A 0.000, B 0.000, C 0.000 }
gfCNCPoint1[4306] = {X 72.7640, Y 64.1739, Z -1.3333, A 0.000, B 0.000, C 0.000 }
gfCNCPoint1[4307] = {X 70.7445, Y 64.2800, Z -1.3333, A 0.000, B 0.000, C 0.000 }
gfCNCPoint1[4308] = {X 64.1851, Y 64.2800, Z -1.3333, A 0.000, B 0.000, C 0.000 }
gfCNCPoint1[4309] = {X 62.0428, Y 64.1606, Z -1.3333, A 0.000, B 0.000, C 0.000 }
gfCNCPoint1[4310] = {X 59.9269, Y 63.8039, Z -1.3333, A 0.000, B 0.000, C 0.000 }
gfCNCPoint1[4311] = {X 57.8638, Y 63.2143, Z -1.3333, A 0.000, B 0.000, C 0.000 }
gfCNCPoint1[4312] = {X 55.8790, Y 62.3991, Z -1.3333, A 0.000, B 0.000, C 0.000 }
gfCNCPoint1[4313] = {X 53.8942, Y 63.2143, Z -1.3333, A 0.000, B 0.000, C 0.000 }
gfCNCPoint1[4314] = {X 51.8311, Y 63.8039, Z -1.3333, A 0.000, B 0.000, C 0.000 }
gfCNCPoint1[4315] = {X 49.7153, Y 64.1606, Z -1.3333, A 0.000, B 0.000, C 0.000 }
gfCNCPoint1[4316] = {X 47.5729, Y 64.2800, Z -1.3333, A 0.000, B 0.000, C 0.000 }
gfCNCPoint1[4317] = {X 40.6393, Y 64.2800, Z -1.3333, A 0.000, B 0.000, C 0.000 }
gfCNCPoint1[4318] = {X 39.1544, Y 64.2227, Z -1.3333, A 0.000, B 0.000, C 0.000 }
gfCNCPoint1[4319] = {X 37.6782, Y 64.0513, Z -1.3333, A 0.000, B 0.000, C 0.000 }
gfCNCPoint1[4320] = {X 36.2197, Y 63.7666, Z -1.3333, A 0.000, B 0.000, C 0.000 }
gfCNCPoint1[4321] = {X 34.1362, Y 64.5931, Z -1.3333, A 0.000, B 0.000, C 0.000 }
gfCNCPoint1[4322] = {X 31.9837, Y 65.2184, Z -1.3333, A 0.000, B 0.000, C 0.000 }
gfCNCPoint1[4323] = {X 29.7817, Y 65.6368, Z -1.3333, A 0.000, B 0.000, C 0.000 }
gfCNCPoint1[4324] = {X 27.0275, Y 66.7154, Z -1.3333, A 0.000, B 0.000, C 0.000 }
gfCNCPoint1[4325] = {X 24.2118, Y 67.6213, Z -1.3333, A 0.000, B 0.000, C 0.000 }
gfCNCPoint1[4326] = {X 23.5941, Y 67.7927, Z -1.3333, A 0.000, B 0.000, C 0.000 }
gfCNCPoint1[4327] = {X 21.3624, Y 68.3451, Z -1.3333, A 0.000, B 0.000, C 0.000 }
gfCNCPoint1[4328] = {X 19.1035, Y 68.7732, Z -1.3333, A 0.000, B 0.000, C 0.000 }
gfCNCPoint1[4329] = {X 19.1035, Y 80.8949, Z -1.3333, A 0.000, B 0.000, C 0.000 }
gfCNCPoint1[4330] = {X 110.5598, Y 80.8949, Z -1.3333, A 0.000, B 0.000, C 0.000 }
gfCNCPoint1[4331] = {X 112.3074, Y 79.4898, Z -1.3333, A 0.000, B 0.000, C 0.000 }
gfCNCPoint1[4332] = {X 114.1908, Y 78.2728, Z -1.3333, A 0.000, B 0.000, C 0.000 }
gfCNCPoint1[4333] = {X 116.1898, Y 77.2568, Z -1.3333, A 0.000, B 0.000, C 0.000 }
gfCNCPoint1[4334] = {X 118.2831, Y 76.4527, Z -1.3333, A 0.000, B 0.000, C 0.000 }
gfCNCPoint1[4335] = {X 133.9641, Y 59.2327, Z -1.3333, A 0.000, B 0.000, C 0.000 }
gfCNCPoint1[4336] = {X 132.7160, Y 58.3551, Z -1.3333, A 0.000, B 0.000, C 0.000 }
gfCNCPoint1[4337] = {X 131.5523, Y 57.3683, Z -1.3333, A 0.000, B 0.000, C 0.000 }
gfCNCPoint1[4338] = {X 130.4824, Y 56.2805, Z -1.3333, A 0.000, B 0.000, C 0.000 }
gfCNCPoint1[4339] = {X 129.6655, Y 55.2988, Z -1.3333, A 0.000, B 0.000, C 0.000 }
gfCNCPoint1[4340] = {X 128.9251, Y 54.2582, Z -1.3333, A 0.000, B 0.000, C 0.000 }
gfCNCPoint1[4341] = {X 128.0750, Y 55.1942, Z -1.3333, A 0.000, B 0.000, C 0.000 }
gfCNCPoint1[4342] = {X 127.1464, Y 56.0525, Z -1.3333, A 0.000, B 0.000, C 0.000 }
gfCNCPoint1[4343] = {X 125.7915, Y 57.0695, Z -1.3333, A 0.000, B 0.000, C 0.000 }
gfCNCPoint1[4344] = {X 124.3270, Y 57.9212, Z -1.3333, A 0.000, B 0.000, C 0.000 }
gfCNCPoint1[4345] = {X 122.7731, Y 58.5961, Z -1.3333, A 0.000, B 0.000, C 0.000 }
gfCNCPoint1[4346] = {X 121.1510, Y 59.0849, Z -1.3333, A 0.000, B 0.000, C 0.000 }
gfCNCPoint1[4347] = {X 119.4828, Y 59.3809, Z -1.3333, A 0.000, B 0.000, C 0.000 }
gfCNCPoint1[4348] = {X 117.7916, Y 59.4800, Z -1.3333, A 0.000, B 0.000, C 0.000 }
gfCNCPoint1[4349] = {X 111.9185, Y 59.4800, Z -1.3333, A 0.000, B 0.000, C 0.000 }
gfCNCPoint1[4350] = {X 111.6599, Y 59.4777, Z -1.3333, A 0.000, B 0.000, C 0.000 }
gfCNCPoint1[4351] = {X 111.4013, Y 59.4708, Z -1.3333, A 0.000, B 0.000, C 0.000 }
gfCNCPoint1[4352] = {X 111.4871, Y 57.0723, Z -1.3333, A 0.000, B 0.000, C 0.000 }
gfCNCPoint1[4353] = {X 109.9587, Y 56.9200, Z -1.3333, A 0.000, B 0.000, C 0.000 }
gfCNCPoint1[4354] = {X 108.4621, Y 56.5750, Z -1.3333, A 0.000, B 0.000, C 0.000 }
gfCNCPoint1[4355] = {X 107.0213, Y 56.0428, Z -1.3333, A 0.000, B 0.000, C 0.000 }
gfCNCPoint1[4356] = {X 105.4432, Y 56.6151, Z -1.3333, A 0.000, B 0.000, C 0.000 }
gfCNCPoint1[4357] = {X 103.8010, Y 56.9630, Z -1.3333, A 0.000, B 0.000, C 0.000 }
gfCNCPoint1[4358] = {X 102.1265, Y 57.0800, Z -1.3333, A 0.000, B 0.000, C 0.000 }
gfCNCPoint1[4359] = {X 100.4519, Y 56.9637, Z -1.3333, A 0.000, B 0.000, C 0.000 }
gfCNCPoint1[4360] = {X 98.8096, Y 56.6164, Z -1.3333, A 0.000, B 0.000, C 0.000 }
gfCNCPoint1[4361] = {X 97.2313, Y 56.0448, Z -1.3333, A 0.000, B 0.000, C 0.000 }
gfCNCPoint1[4362] = {X 95.6538, Y 56.6162, Z -1.3333, A 0.000, B 0.000, C 0.000 }
gfCNCPoint1[4363] = {X 94.0123, Y 56.9635, Z -1.3333, A 0.000, B 0.000, C 0.000 }
gfCNCPoint1[4364] = {X 92.3385, Y 57.0800, Z -1.3333, A 0.000, B 0.000, C 0.000 }
gfCNCPoint1[4365] = {X 85.8951, Y 57.0800, Z -1.3333, A 0.000, B 0.000, C 0.000 }
gfCNCPoint1[4366] = {X 84.3894, Y 56.9858, Z -1.3333, A 0.000, B 0.000, C 0.000 }
gfCNCPoint1[4367] = {X 82.9073, Y 56.7047, Z -1.3333, A 0.000, B 0.000, C 0.000 }
gfCNCPoint1[4368] = {X 81.4847, Y 58.0224, Z -1.3333, A 0.000, B 0.000, C 0.000 }
gfCNCPoint1[4369] = {X 79.9203, Y 59.1682, Z -1.3333, A 0.000, B 0.000, C 0.000 }
gfCNCPoint1[4370] = {X 78.2348, Y 60.1271, Z -1.3333, A 0.000, B 0.000, C 0.000 }
gfCNCPoint1[4371] = {X 76.4504, Y 60.8864, Z -1.3333, A 0.000, B 0.000, C 0.000 }
gfCNCPoint1[4372] = {X 74.5908, Y 61.4359, Z -1.3333, A 0.000, B 0.000, C 0.000 }
gfCNCPoint1[4373] = {X 72.6804, Y 61.7686, Z -1.3333, A 0.000, B 0.000, C 0.000 }
gfCNCPoint1[4374] = {X 70.7445, Y 61.8800, Z -1.3333, A 0.000, B 0.000, C 0.000 }
gfCNCPoint1[4375] = {X 64.1851, Y 61.8800, Z -1.3333, A 0.000, B 0.000, C 0.000 }
gfCNCPoint1[4376] = {X 62.4514, Y 61.7907, Z -1.3333, A 0.000, B 0.000, C 0.000 }
gfCNCPoint1[4377] = {X 60.7359, Y 61.5238, Z -1.3333, A 0.000, B 0.000, C 0.000 }
gfCNCPoint1[4378] = {X 59.0570, Y 61.0822, Z -1.3333, A 0.000, B 0.000, C 0.000 }
gfCNCPoint1[4379] = {X 57.4323, Y 60.4704, Z -1.3333, A 0.000, B 0.000, C 0.000 }
gfCNCPoint1[4380] = {X 55.8790, Y 59.6950, Z -1.3333, A 0.000, B 0.000, C 0.000 }
gfCNCPoint1[4381] = {X 54.3258, Y 60.4704, Z -1.3333, A 0.000, B 0.000, C 0.000 }
gfCNCPoint1[4382] = {X 52.7011, Y 61.0822, Z -1.3333, A 0.000, B 0.000, C 0.000 }
gfCNCPoint1[4383] = {X 51.0221, Y 61.5238, Z -1.3333, A 0.000, B 0.000, C 0.000 }
gfCNCPoint1[4384] = {X 49.3067, Y 61.7907, Z -1.3333, A 0.000, B 0.000, C 0.000 }
gfCNCPoint1[4385] = {X 47.5729, Y 61.8800, Z -1.3333, A 0.000, B 0.000, C 0.000 }
gfCNCPoint1[4386] = {X 40.6393, Y 61.8800, Z -1.3333, A 0.000, B 0.000, C 0.000 }
gfCNCPoint1[4387] = {X 39.0674, Y 61.8067, Z -1.3333, A 0.000, B 0.000, C 0.000 }
gfCNCPoint1[4388] = {X 37.5092, Y 61.5872, Z -1.3333, A 0.000, B 0.000, C 0.000 }
gfCNCPoint1[4389] = {X 35.9782, Y 61.2237, Z -1.3333, A 0.000, B 0.000, C 0.000 }
gfCNCPoint1[4390] = {X 34.3395, Y 61.9591, Z -1.3333, A 0.000, B 0.000, C 0.000 }
gfCNCPoint1[4391] = {X 32.6445, Y 62.5533, Z -1.3333, A 0.000, B 0.000, C 0.000 }
gfCNCPoint1[4392] = {X 30.9053, Y 63.0020, Z -1.3333, A 0.000, B 0.000, C 0.000 }
gfCNCPoint1[4393] = {X 29.1344, Y 63.3020, Z -1.3333, A 0.000, B 0.000, C 0.000 }
gfCNCPoint1[4394] = {X 26.3794, Y 64.3982, Z -1.3333, A 0.000, B 0.000, C 0.000 }
gfCNCPoint1[4395] = {X 23.5587, Y 65.3119, Z -1.3333, A 0.000, B 0.000, C 0.000 }
gfCNCPoint1[4396] = {X 22.9533, Y 65.4799, Z -1.3333, A 0.000, B 0.000, C 0.000 }
gfCNCPoint1[4397] = {X 20.8927, Y 65.9911, Z -1.3333, A 0.000, B 0.000, C 0.000 }
gfCNCPoint1[4398] = {X 18.8074, Y 66.3898, Z -1.3333, A 0.000, B 0.000, C 0.000 }
gfCNCPoint1[4399] = {X 16.7035, Y 66.6749, Z -1.3333, A 0.000, B 0.000, C 0.000 }
gfCNCPoint1[4400] = {X 16.7035, Y 83.2949, Z -1.3333, A 0.000, B 0.000, C 0.000 }
gfCNCPoint1[4401] = {X 111.5064, Y 83.2949, Z -1.3333, A 0.000, B 0.000, C 0.000 }
gfCNCPoint1[4402] = {X 112.9253, Y 82.0353, Z -1.3333, A 0.000, B 0.000, C 0.000 }
gfCNCPoint1[4403] = {X 114.4611, Y 80.9213, Z -1.3333, A 0.000, B 0.000, C 0.000 }
gfCNCPoint1[4404] = {X 116.0990, Y 79.9636, Z -1.3333, A 0.000, B 0.000, C 0.000 }
gfCNCPoint1[4405] = {X 117.8231, Y 79.1715, Z -1.3333, A 0.000, B 0.000, C 0.000 }
gfCNCPoint1[4406] = {X 119.6167, Y 78.5527, Z -1.3333, A 0.000, B 0.000, C 0.000 }
gfCNCPoint1[4407] = {X 137.8581, Y 58.5212, Z -1.3333, A 0.000, B 0.000, C 0.000 }
gfCNCPoint1[4408] = {X 136.5232, Y 57.9308, Z -1.3333, A 0.000, B 0.000, C 0.000 }
gfCNCPoint1[4409] = {X 135.2545, Y 57.2091, Z -1.3333, A 0.000, B 0.000, C 0.000 }
gfCNCPoint1[4410] = {X 134.0104, Y 56.3200, Z -1.3333, A 0.000, B 0.000, C 0.000 }
gfCNCPoint1[4411] = {X 132.8669, Y 55.3047, Z -1.3333, A 0.000, B 0.000, C 0.000 }
gfCNCPoint1[4412] = {X 131.8370, Y 54.1745, Z -1.3333, A 0.000, B 0.000, C 0.000 }
gfCNCPoint1[4413] = {X 130.9319, Y 52.9419, Z -1.3333, A 0.000, B 0.000, C 0.000 }
gfCNCPoint1[4414] = {X 130.2147, Y 51.7225, Z -1.3333, A 0.000, B 0.000, C 0.000 }
gfCNCPoint1[4415] = {X 129.6199, Y 50.4390, Z -1.3333, A 0.000, B 0.000, C 0.000 }
gfCNCPoint1[4416] = {X 129.1532, Y 49.1035, Z -1.3333, A 0.000, B 0.000, C 0.000 }
gfCNCPoint1[4417] = {X 128.6036, Y 50.3877, Z -1.3333, A 0.000, B 0.000, C 0.000 }
gfCNCPoint1[4418] = {X 127.9093, Y 51.5998, Z -1.3333, A 0.000, B 0.000, C 0.000 }
gfCNCPoint1[4419] = {X 127.0798, Y 52.7237, Z -1.3333, A 0.000, B 0.000, C 0.000 }
gfCNCPoint1[4420] = {X 126.0417, Y 53.8239, Z -1.3333, A 0.000, B 0.000, C 0.000 }
gfCNCPoint1[4421] = {X 124.8743, Y 54.7858, Z -1.3333, A 0.000, B 0.000, C 0.000 }
gfCNCPoint1[4422] = {X 123.5958, Y 55.5942, Z -1.3333, A 0.000, B 0.000, C 0.000 }
gfCNCPoint1[4423] = {X 122.2263, Y 56.2365, Z -1.3333, A 0.000, B 0.000, C 0.000 }
gfCNCPoint1[4424] = {X 120.7872, Y 56.7027, Z -1.3333, A 0.000, B 0.000, C 0.000 }
gfCNCPoint1[4425] = {X 119.3012, Y 56.9853, Z -1.3333, A 0.000, B 0.000, C 0.000 }
gfCNCPoint1[4426] = {X 117.7916, Y 57.0800, Z -1.3333, A 0.000, B 0.000, C 0.000 }
gfCNCPoint1[4427] = {X 111.9185, Y 57.0800, Z -1.3333, A 0.000, B 0.000, C 0.000 }
gfCNCPoint1[4428] = {X 111.7027, Y 57.0781, Z -1.3333, A 0.000, B 0.000, C 0.000 }
gfCNCPoint1[4429] = {X 111.4871, Y 57.0723, Z -1.3333, A 0.000, B 0.000, C 0.000 }
gfCNCPoint1[4430] = {X 111.5728, Y 54.6738, Z -1.3333, A 0.000, B 0.000, C 0.000 }
gfCNCPoint1[4431] = {X 110.3820, Y 54.5573, Z -1.3333, A 0.000, B 0.000, C 0.000 }
gfCNCPoint1[4432] = {X 109.2147, Y 54.2947, Z -1.3333, A 0.000, B 0.000, C 0.000 }
gfCNCPoint1[4433] = {X 108.0887, Y 53.8902, Z -1.3333, A 0.000, B 0.000, C 0.000 }
gfCNCPoint1[4434] = {X 107.0213, Y 53.3498, Z -1.3333, A 0.000, B 0.000, C 0.000 }
gfCNCPoint1[4435] = {X 106.6480, Y 53.5578, Z -1.3333, A 0.000, B 0.000, C 0.000 }
gfCNCPoint1[4436] = {X 106.2658, Y 53.7492, Z -1.3333, A 0.000, B 0.000, C 0.000 }
gfCNCPoint1[4437] = {X 105.0149, Y 54.2383, Z -1.3333, A 0.000, B 0.000, C 0.000 }
gfCNCPoint1[4438] = {X 103.7084, Y 54.5495, Z -1.3333, A 0.000, B 0.000, C 0.000 }
gfCNCPoint1[4439] = {X 102.3713, Y 54.6768, Z -1.3333, A 0.000, B 0.000, C 0.000 }
gfCNCPoint1[4440] = {X 101.0295, Y 54.6179, Z -1.3333, A 0.000, B 0.000, C 0.000 }
gfCNCPoint1[4441] = {X 99.7088, Y 54.3738, Z -1.3333, A 0.000, B 0.000, C 0.000 }
gfCNCPoint1[4442] = {X 98.4345, Y 53.9493, Z -1.3333, A 0.000, B 0.000, C 0.000 }
gfCNCPoint1[4443] = {X 97.2313, Y 53.3524, Z -1.3333, A 0.000, B 0.000, C 0.000 }
gfCNCPoint1[4444] = {X 96.0852, Y 53.9255, Z -1.3333, A 0.000, B 0.000, C 0.000 }
gfCNCPoint1[4445] = {X 94.8734, Y 54.3422, Z -1.3333, A 0.000, B 0.000, C 0.000 }
gfCNCPoint1[4446] = {X 93.6172, Y 54.5952, Z -1.3333, A 0.000, B 0.000, C 0.000 }
gfCNCPoint1[4447] = {X 92.3385, Y 54.6800, Z -1.3333, A 0.000, B 0.000, C 0.000 }
gfCNCPoint1[4448] = {X 85.8951, Y 54.6800, Z -1.3333, A 0.000, B 0.000, C 0.000 }
gfCNCPoint1[4449] = {X 84.6159, Y 54.5951, Z -1.3333, A 0.000, B 0.000, C 0.000 }
gfCNCPoint1[4450] = {X 83.3592, Y 54.3419, Z -1.3333, A 0.000, B 0.000, C 0.000 }
gfCNCPoint1[4451] = {X 82.1469, Y 53.9249, Z -1.3333, A 0.000, B 0.000, C 0.000 }
gfCNCPoint1[4452] = {X 81.0644, Y 55.1572, Z -1.3333, A 0.000, B 0.000, C 0.000 }
gfCNCPoint1[4453] = {X 79.8495, Y 56.2591, Z -1.3333, A 0.000, B 0.000, C 0.000 }
gfCNCPoint1[4454] = {X 78.5178, Y 57.2166, Z -1.3333, A 0.000, B 0.000, C 0.000 }
gfCNCPoint1[4455] = {X 77.0863, Y 58.0174, Z -1.3333, A 0.000, B 0.000, C 0.000 }
gfCNCPoint1[4456] = {X 75.5734, Y 58.6511, Z -1.3333, A 0.000, B 0.000, C 0.000 }
gfCNCPoint1[4457] = {X 73.9986, Y 59.1096, Z -1.3333, A 0.000, B 0.000, C 0.000 }
gfCNCPoint1[4458] = {X 72.3820, Y 59.3871, Z -1.3333, A 0.000, B 0.000, C 0.000 }
gfCNCPoint1[4459] = {X 70.7445, Y 59.4800, Z -1.3333, A 0.000, B 0.000, C 0.000 }
gfCNCPoint1[4460] = {X 64.1851, Y 59.4800, Z -1.3333, A 0.000, B 0.000, C 0.000 }
gfCNCPoint1[4461] = {X 62.4203, Y 59.3720, Z -1.3333, A 0.000, B 0.000, C 0.000 }
gfCNCPoint1[4462] = {X 60.6818, Y 59.0498, Z -1.3333, A 0.000, B 0.000, C 0.000 }
gfCNCPoint1[4463] = {X 58.9955, Y 58.5181, Z -1.3333, A 0.000, B 0.000, C 0.000 }
gfCNCPoint1[4464] = {X 57.3866, Y 57.7848, Z -1.3333, A 0.000, B 0.000, C 0.000 }
gfCNCPoint1[4465] = {X 55.8790, Y 56.8608, Z -1.3333, A 0.000, B 0.000, C 0.000 }
gfCNCPoint1[4466] = {X 54.3715, Y 57.7848, Z -1.3333, A 0.000, B 0.000, C 0.000 }
gfCNCPoint1[4467] = {X 52.7626, Y 58.5181, Z -1.3333, A 0.000, B 0.000, C 0.000 }
gfCNCPoint1[4468] = {X 51.0763, Y 59.0498, Z -1.3333, A 0.000, B 0.000, C 0.000 }
gfCNCPoint1[4469] = {X 49.3378, Y 59.3720, Z -1.3333, A 0.000, B 0.000, C 0.000 }
gfCNCPoint1[4470] = {X 47.5729, Y 59.4800, Z -1.3333, A 0.000, B 0.000, C 0.000 }
gfCNCPoint1[4471] = {X 40.6393, Y 59.4800, Z -1.3333, A 0.000, B 0.000, C 0.000 }
gfCNCPoint1[4472] = {X 38.9794, Y 59.3845, Z -1.3333, A 0.000, B 0.000, C 0.000 }
gfCNCPoint1[4473] = {X 37.3414, Y 59.0994, Z -1.3333, A 0.000, B 0.000, C 0.000 }
gfCNCPoint1[4474] = {X 35.7468, Y 58.6284, Z -1.3333, A 0.000, B 0.000, C 0.000 }
gfCNCPoint1[4475] = {X 34.0329, Y 59.4861, Z -1.3333, A 0.000, B 0.000, C 0.000 }
gfCNCPoint1[4476] = {X 32.2407, Y 60.1651, Z -1.3333, A 0.000, B 0.000, C 0.000 }
gfCNCPoint1[4477] = {X 30.3887, Y 60.6582, Z -1.3333, A 0.000, B 0.000, C 0.000 }
gfCNCPoint1[4478] = {X 28.4962, Y 60.9604, Z -1.3333, A 0.000, B 0.000, C 0.000 }
gfCNCPoint1[4479] = {X 25.7362, Y 62.0785, Z -1.3333, A 0.000, B 0.000, C 0.000 }
gfCNCPoint1[4480] = {X 22.9052, Y 63.0025, Z -1.3333, A 0.000, B 0.000, C 0.000 }
gfCNCPoint1[4481] = {X 22.3124, Y 63.1670, Z -1.3333, A 0.000, B 0.000, C 0.000 }
gfCNCPoint1[4482] = {X 19.6769, Y 63.7937, Z -1.3333, A 0.000, B 0.000, C 0.000 }
gfCNCPoint1[4483] = {X 17.0025, Y 64.2244, Z -1.3333, A 0.000, B 0.000, C 0.000 }
gfCNCPoint1[4484] = {X 14.3035, Y 64.4570, Z -1.3333, A 0.000, B 0.000, C 0.000 }
gfCNCPoint1[4485] = {X 14.3035, Y 85.6949, Z -1.3333, A 0.000, B 0.000, C 0.000 }
gfCNCPoint1[4486] = {X 112.5247, Y 85.6949, Z -1.3333, A 0.000, B 0.000, C 0.000 }
gfCNCPoint1[4487] = {X 113.9438, Y 84.3108, Z -1.3333, A 0.000, B 0.000, C 0.000 }
gfCNCPoint1[4488] = {X 115.5154, Y 83.1025, Z -1.3333, A 0.000, B 0.000, C 0.000 }
gfCNCPoint1[4489] = {X 117.2178, Y 82.0869, Z -1.3333, A 0.000, B 0.000, C 0.000 }
gfCNCPoint1[4490] = {X 119.0275, Y 81.2779, Z -1.3333, A 0.000, B 0.000, C 0.000 }
gfCNCPoint1[4491] = {X 120.9196, Y 80.6865, Z -1.3333, A 0.000, B 0.000, C 0.000 }
gfCNCPoint1[4492] = {X 142.4305, Y 57.0646, Z -1.3333, A 0.000, B 0.000, C 0.000 }
gfCNCPoint1[4493] = {X 141.1673, Y 56.9340, Z -1.3333, A 0.000, B 0.000, C 0.000 }
gfCNCPoint1[4494] = {X 139.9249, Y 56.6715, Z -1.3333, A 0.000, B 0.000, C 0.000 }
gfCNCPoint1[4495] = {X 138.7169, Y 56.2801, Z -1.3333, A 0.000, B 0.000, C 0.000 }
gfCNCPoint1[4496] = {X 137.2797, Y 55.6184, Z -1.3333, A 0.000, B 0.000, C 0.000 }
gfCNCPoint1[4497] = {X 135.9413, Y 54.7745, Z -1.3333, A 0.000, B 0.000, C 0.000 }
gfCNCPoint1[4498] = {X 134.7247, Y 53.7629, Z -1.3333, A 0.000, B 0.000, C 0.000 }
gfCNCPoint1[4499] = {X 133.6507, Y 52.6010, Z -1.3333, A 0.000, B 0.000, C 0.000 }
gfCNCPoint1[4500] = {X 132.7378, Y 51.3087, Z -1.3333, A 0.000, B 0.000, C 0.000 }
gfCNCPoint1[4501] = {X 132.0017, Y 49.9081, Z -1.3333, A 0.000, B 0.000, C 0.000 }
gfCNCPoint1[4502] = {X 131.4549, Y 48.4234, Z -1.3333, A 0.000, B 0.000, C 0.000 }
gfCNCPoint1[4503] = {X 131.1845, Y 47.3200, Z -1.3333, A 0.000, B 0.000, C 0.000 }
gfCNCPoint1[4504] = {X 131.0190, Y 46.1961, Z -1.3333, A 0.000, B 0.000, C 0.000 }
gfCNCPoint1[4505] = {X 130.9598, Y 45.0616, Z -1.3333, A 0.000, B 0.000, C 0.000 }
gfCNCPoint1[4506] = {X 130.9601, Y 44.0978, Z -1.3333, A 0.000, B 0.000, C 0.000 }
gfCNCPoint1[4507] = {X 131.0921, Y 42.4244, Z -1.3333, A 0.000, B 0.000, C 0.000 }
gfCNCPoint1[4508] = {X 131.4548, Y 40.7854, Z -1.3333, A 0.000, B 0.000, C 0.000 }
gfCNCPoint1[4509] = {X 133.7565, Y 41.4655, Z -1.3333, A 0.000, B 0.000, C 0.000 }
gfCNCPoint1[4510] = {X 134.2330, Y 40.1906, Z -1.3333, A 0.000, B 0.000, C 0.000 }
gfCNCPoint1[4511] = {X 134.8836, Y 38.9952, Z -1.3333, A 0.000, B 0.000, C 0.000 }
gfCNCPoint1[4512] = {X 134.8836, Y 27.0854, Z -1.3333, A 0.000, B 0.000, C 0.000 }
gfCNCPoint1[4513] = {X 134.3931, Y 27.1259, Z -1.3333, A 0.000, B 0.000, C 0.000 }
gfCNCPoint1[4514] = {X 133.9011, Y 27.1414, Z -1.3333, A 0.000, B 0.000, C 0.000 }
gfCNCPoint1[4515] = {X 133.2006, Y 27.1415, Z -1.3333, A 0.000, B 0.000, C 0.000 }
gfCNCPoint1[4516] = {X 131.9565, Y 27.0612, Z -1.3333, A 0.000, B 0.000, C 0.000 }
gfCNCPoint1[4517] = {X 130.7329, Y 26.8217, Z -1.3333, A 0.000, B 0.000, C 0.000 }
gfCNCPoint1[4518] = {X 129.5503, Y 26.4269, Z -1.3333, A 0.000, B 0.000, C 0.000 }
gfCNCPoint1[4519] = {X 128.4282, Y 25.8833, Z -1.3333, A 0.000, B 0.000, C 0.000 }
gfCNCPoint1[4520] = {X 127.3853, Y 25.2001, Z -1.3333, A 0.000, B 0.000, C 0.000 }
gfCNCPoint1[4521] = {X 126.3431, Y 24.2936, Z -1.3333, A 0.000, B 0.000, C 0.000 }
gfCNCPoint1[4522] = {X 125.4406, Y 23.2480, Z -1.3333, A 0.000, B 0.000, C 0.000 }
gfCNCPoint1[4523] = {X 124.6960, Y 22.0847, Z -1.3333, A 0.000, B 0.000, C 0.000 }
gfCNCPoint1[4524] = {X 124.1246, Y 20.8271, Z -1.3333, A 0.000, B 0.000, C 0.000 }
gfCNCPoint1[4525] = {X 123.7379, Y 19.5011, Z -1.3333, A 0.000, B 0.000, C 0.000 }
gfCNCPoint1[4526] = {X 123.5440, Y 18.1335, Z -1.3333, A 0.000, B 0.000, C 0.000 }
gfCNCPoint1[4527] = {X 123.5429, Y 39.7455, Z -1.3333, A 0.000, B 0.000, C 0.000 }
gfCNCPoint1[4528] = {X 124.1919, Y 40.7397, Z -1.3333, A 0.000, B 0.000, C 0.000 }
gfCNCPoint1[4529] = {X 124.6707, Y 41.8262, Z -1.3333, A 0.000, B 0.000, C 0.000 }
gfCNCPoint1[4530] = {X 124.9665, Y 42.9761, Z -1.3333, A 0.000, B 0.000, C 0.000 }
gfCNCPoint1[4531] = {X 125.0714, Y 44.1587, Z -1.3333, A 0.000, B 0.000, C 0.000 }
gfCNCPoint1[4532] = {X 125.0716, Y 45.0000, Z -1.3333, A 0.000, B 0.000, C 0.000 }
gfCNCPoint1[4533] = {X 124.9610, Y 46.2642, Z -1.3333, A 0.000, B 0.000, C 0.000 }
gfCNCPoint1[4534] = {X 124.6325, Y 47.4899, Z -1.3333, A 0.000, B 0.000, C 0.000 }
gfCNCPoint1[4535] = {X 124.0962, Y 48.6400, Z -1.3333, A 0.000, B 0.000, C 0.000 }
gfCNCPoint1[4536] = {X 123.3684, Y 49.6795, Z -1.3333, A 0.000, B 0.000, C 0.000 }
gfCNCPoint1[4537] = {X 122.4711, Y 50.5768, Z -1.3333, A 0.000, B 0.000, C 0.000 }
gfCNCPoint1[4538] = {X 121.4316, Y 51.3047, Z -1.3333, A 0.000, B 0.000, C 0.000 }
gfCNCPoint1[4539] = {X 120.2815, Y 51.8410, Z -1.3333, A 0.000, B 0.000, C 0.000 }
gfCNCPoint1[4540] = {X 119.0557, Y 52.1694, Z -1.3333, A 0.000, B 0.000, C 0.000 }
gfCNCPoint1[4541] = {X 117.7916, Y 52.2800, Z -1.3333, A 0.000, B 0.000, C 0.000 }
gfCNCPoint1[4542] = {X 111.9185, Y 52.2800, Z -1.3333, A 0.000, B 0.000, C 0.000 }
gfCNCPoint1[4543] = {X 110.8481, Y 52.2009, Z -1.3333, A 0.000, B 0.000, C 0.000 }
gfCNCPoint1[4544] = {X 109.8009, Y 51.9652, Z -1.3333, A 0.000, B 0.000, C 0.000 }
gfCNCPoint1[4545] = {X 108.7998, Y 51.5782, Z -1.3333, A 0.000, B 0.000, C 0.000 }
gfCNCPoint1[4546] = {X 107.8665, Y 51.0481, Z -1.3333, A 0.000, B 0.000, C 0.000 }
gfCNCPoint1[4547] = {X 107.0213, Y 50.3866, Z -1.3333, A 0.000, B 0.000, C 0.000 }
gfCNCPoint1[4548] = {X 106.1743, Y 51.0493, Z -1.3333, A 0.000, B 0.000, C 0.000 }
gfCNCPoint1[4549] = {X 105.2389, Y 51.5800, Z -1.3333, A 0.000, B 0.000, C 0.000 }
gfCNCPoint1[4550] = {X 104.0917, Y 52.0091, Z -1.3333, A 0.000, B 0.000, C 0.000 }
gfCNCPoint1[4551] = {X 102.8887, Y 52.2397, Z -1.3333, A 0.000, B 0.000, C 0.000 }
gfCNCPoint1[4552] = {X 101.6641, Y 52.2655, Z -1.3333, A 0.000, B 0.000, C 0.000 }
gfCNCPoint1[4553] = {X 100.4526, Y 52.0855, Z -1.3333, A 0.000, B 0.000, C 0.000 }
gfCNCPoint1[4554] = {X 99.2883, Y 51.7050, Z -1.3333, A 0.000, B 0.000, C 0.000 }
gfCNCPoint1[4555] = {X 98.2043, Y 51.1347, Z -1.3333, A 0.000, B 0.000, C 0.000 }
gfCNCPoint1[4556] = {X 97.2313, Y 50.3907, Z -1.3333, A 0.000, B 0.000, C 0.000 }
gfCNCPoint1[4557] = {X 96.3865, Y 51.0508, Z -1.3333, A 0.000, B 0.000, C 0.000 }
gfCNCPoint1[4558] = {X 95.4539, Y 51.5797, Z -1.3333, A 0.000, B 0.000, C 0.000 }
gfCNCPoint1[4559] = {X 94.4538, Y 51.9659, Z -1.3333, A 0.000, B 0.000, C 0.000 }
gfCNCPoint1[4560] = {X 93.4078, Y 52.2011, Z -1.3333, A 0.000, B 0.000, C 0.000 }
gfCNCPoint1[4561] = {X 92.3385, Y 52.2800, Z -1.3333, A 0.000, B 0.000, C 0.000 }
gfCNCPoint1[4562] = {X 85.8951, Y 52.2800, Z -1.3333, A 0.000, B 0.000, C 0.000 }
gfCNCPoint1[4563] = {X 84.6852, Y 52.1788, Z -1.3333, A 0.000, B 0.000, C 0.000 }
gfCNCPoint1[4564] = {X 83.5090, Y 51.8779, Z -1.3333, A 0.000, B 0.000, C 0.000 }
gfCNCPoint1[4565] = {X 82.3992, Y 51.3857, Z -1.3333, A 0.000, B 0.000, C 0.000 }
gfCNCPoint1[4566] = {X 81.3866, Y 50.7159, Z -1.3333, A 0.000, B 0.000, C 0.000 }
gfCNCPoint1[4567] = {X 80.5223, Y 52.0937, Z -1.3333, A 0.000, B 0.000, C 0.000 }
gfCNCPoint1[4568] = {X 79.4808, Y 53.3429, Z -1.3333, A 0.000, B 0.000, C 0.000 }
gfCNCPoint1[4569] = {X 78.2809, Y 54.4408, Z -1.3333, A 0.000, B 0.000, C 0.000 }
gfCNCPoint1[4570] = {X 76.9444, Y 55.3676, Z -1.3333, A 0.000, B 0.000, C 0.000 }
gfCNCPoint1[4571] = {X 75.4955, Y 56.1065, Z -1.3333, A 0.000, B 0.000, C 0.000 }
gfCNCPoint1[4572] = {X 73.9605, Y 56.6440, Z -1.3333, A 0.000, B 0.000, C 0.000 }
gfCNCPoint1[4573] = {X 72.3672, Y 56.9705, Z -1.3333, A 0.000, B 0.000, C 0.000 }
gfCNCPoint1[4574] = {X 70.7445, Y 57.0800, Z -1.3333, A 0.000, B 0.000, C 0.000 }
gfCNCPoint1[4575] = {X 64.1851, Y 57.0800, Z -1.3333, A 0.000, B 0.000, C 0.000 }
gfCNCPoint1[4576] = {X 62.6628, Y 56.9837, Z -1.3333, A 0.000, B 0.000, C 0.000 }
gfCNCPoint1[4577] = {X 61.1646, Y 56.6963, Z -1.3333, A 0.000, B 0.000, C 0.000 }
gfCNCPoint1[4578] = {X 59.7147, Y 56.2224, Z -1.3333, A 0.000, B 0.000, C 0.000 }
gfCNCPoint1[4579] = {X 58.3360, Y 55.5695, Z -1.3333, A 0.000, B 0.000, C 0.000 }
gfCNCPoint1[4580] = {X 57.0507, Y 54.7481, Z -1.3333, A 0.000, B 0.000, C 0.000 }
gfCNCPoint1[4581] = {X 55.8790, Y 53.7713, Z -1.3333, A 0.000, B 0.000, C 0.000 }
gfCNCPoint1[4582] = {X 54.7074, Y 54.7481, Z -1.3333, A 0.000, B 0.000, C 0.000 }
gfCNCPoint1[4583] = {X 53.4220, Y 55.5695, Z -1.3333, A 0.000, B 0.000, C 0.000 }
gfCNCPoint1[4584] = {X 52.0434, Y 56.2224, Z -1.3333, A 0.000, B 0.000, C 0.000 }
gfCNCPoint1[4585] = {X 50.5934, Y 56.6963, Z -1.3333, A 0.000, B 0.000, C 0.000 }
gfCNCPoint1[4586] = {X 49.0953, Y 56.9837, Z -1.3333, A 0.000, B 0.000, C 0.000 }
gfCNCPoint1[4587] = {X 47.5729, Y 57.0800, Z -1.3333, A 0.000, B 0.000, C 0.000 }
gfCNCPoint1[4588] = {X 40.6393, Y 57.0800, Z -1.3333, A 0.000, B 0.000, C 0.000 }
gfCNCPoint1[4589] = {X 39.3237, Y 57.0081, Z -1.3333, A 0.000, B 0.000, C 0.000 }
gfCNCPoint1[4590] = {X 38.0237, Y 56.7934, Z -1.3333, A 0.000, B 0.000, C 0.000 }
gfCNCPoint1[4591] = {X 36.7548, Y 56.4384, Z -1.3333, A 0.000, B 0.000, C 0.000 }
gfCNCPoint1[4592] = {X 35.5321, Y 55.9473, Z -1.3333, A 0.000, B 0.000, C 0.000 }
gfCNCPoint1[4593] = {X 34.1217, Y 56.7815, Z -1.3333, A 0.000, B 0.000, C 0.000 }
gfCNCPoint1[4594] = {X 32.6352, Y 57.4709, Z -1.3333, A 0.000, B 0.000, C 0.000 }
gfCNCPoint1[4595] = {X 31.0874, Y 58.0088, Z -1.3333, A 0.000, B 0.000, C 0.000 }
gfCNCPoint1[4596] = {X 29.4936, Y 58.3897, Z -1.3333, A 0.000, B 0.000, C 0.000 }
gfCNCPoint1[4597] = {X 27.8699, Y 58.6098, Z -1.3333, A 0.000, B 0.000, C 0.000 }
gfCNCPoint1[4598] = {X 25.0992, Y 59.7555, Z -1.3333, A 0.000, B 0.000, C 0.000 }
gfCNCPoint1[4599] = {X 22.2515, Y 60.6932, Z -1.3333, A 0.000, B 0.000, C 0.000 }
gfCNCPoint1[4600] = {X 21.6715, Y 60.8542, Z -1.3333, A 0.000, B 0.000, C 0.000 }
gfCNCPoint1[4601] = {X 19.2694, Y 61.4276, Z -1.3333, A 0.000, B 0.000, C 0.000 }
gfCNCPoint1[4602] = {X 16.8323, Y 61.8270, Z -1.3333, A 0.000, B 0.000, C 0.000 }
gfCNCPoint1[4603] = {X 14.3728, Y 62.0502, Z -1.3333, A 0.000, B 0.000, C 0.000 }
gfCNCPoint1[4604] = {X 11.9035, Y 62.0960, Z -1.3333, A 0.000, B 0.000, C 0.000 }
gfCNCPoint1[4605] = {X 11.9035, Y 88.0949, Z -1.3333, A 0.000, B 0.000, C 0.000 }
gfCNCPoint1[4606] = {X 113.6338, Y 88.0949, Z -1.3333, A 0.000, B 0.000, C 0.000 }
gfCNCPoint1[4607] = {X 114.7671, Y 86.8210, Z -1.3333, A 0.000, B 0.000, C 0.000 }
gfCNCPoint1[4608] = {X 116.0423, Y 85.6892, Z -1.3333, A 0.000, B 0.000, C 0.000 }
gfCNCPoint1[4609] = {X 117.4418, Y 84.7151, Z -1.3333, A 0.000, B 0.000, C 0.000 }
gfCNCPoint1[4610] = {X 118.9460, Y 83.9123, Z -1.3333, A 0.000, B 0.000, C 0.000 }
gfCNCPoint1[4611] = {X 120.5341, Y 83.2918, Z -1.3333, A 0.000, B 0.000, C 0.000 }
gfCNCPoint1[4612] = {X 122.1842, Y 82.8624, Z -1.3333, A 0.000, B 0.000, C 0.000 }
gfCNCPoint1[4613] = {X 144.8180, Y 58.0074, Z -1.3333, A 0.000, B 0.000, C 0.000 }
gfCNCPoint1[4614] = {X 144.9143, Y 56.3325, Z -1.3333, A 0.000, B 0.000, C 0.000 }
gfCNCPoint1[4615] = {X 145.2037, Y 54.6800, Z -1.3333, A 0.000, B 0.000, C 0.000 }
gfCNCPoint1[4616] = {X 143.0396, Y 54.6800, Z -1.3333, A 0.000, B 0.000, C 0.000 }
gfCNCPoint1[4617] = {X 142.7955, Y 54.6769, Z -1.3333, A 0.000, B 0.000, C 0.000 }
gfCNCPoint1[4618] = {X 142.5515, Y 54.6677, Z -1.3333, A 0.000, B 0.000, C 0.000 }
gfCNCPoint1[4619] = {X 141.0984, Y 54.4833, Z -1.3333, A 0.000, B 0.000, C 0.000 }
gfCNCPoint1[4620] = {X 139.6897, Y 54.0819, Z -1.3333, A 0.000, B 0.000, C 0.000 }
gfCNCPoint1[4621] = {X 138.3577, Y 53.4724, Z -1.3333, A 0.000, B 0.000, C 0.000 }
gfCNCPoint1[4622] = {X 137.1329, Y 52.6690, Z -1.3333, A 0.000, B 0.000, C 0.000 }
gfCNCPoint1[4623] = {X 136.0434, Y 51.6899, Z -1.3333, A 0.000, B 0.000, C 0.000 }
gfCNCPoint1[4624] = {X 135.1141, Y 50.5577, Z -1.3333, A 0.000, B 0.000, C 0.000 }
gfCNCPoint1[4625] = {X 134.3662, Y 49.2982, Z -1.3333, A 0.000, B 0.000, C 0.000 }
gfCNCPoint1[4626] = {X 133.8170, Y 47.9403, Z -1.3333, A 0.000, B 0.000, C 0.000 }
gfCNCPoint1[4627] = {X 133.4789, Y 46.5151, Z -1.3333, A 0.000, B 0.000, C 0.000 }
gfCNCPoint1[4628] = {X 133.3598, Y 45.0552, Z -1.3333, A 0.000, B 0.000, C 0.000 }
gfCNCPoint1[4629] = {X 133.3601, Y 44.1104, Z -1.3333, A 0.000, B 0.000, C 0.000 }
gfCNCPoint1[4630] = {X 133.4665, Y 42.7742, Z -1.3333, A 0.000, B 0.000, C 0.000 }
gfCNCPoint1[4631] = {X 133.7565, Y 41.4655, Z -1.3333, A 0.000, B 0.000, C 0.000 }
gfCNCPoint1[4632] = {X 136.0581, Y 42.1457, Z -1.3333, A 0.000, B 0.000, C 0.000 }
gfCNCPoint1[4633] = {X 136.3664, Y 41.2990, Z -1.3333, A 0.000, B 0.000, C 0.000 }
gfCNCPoint1[4634] = {X 136.7770, Y 40.4969, Z -1.3333, A 0.000, B 0.000, C 0.000 }
gfCNCPoint1[4635] = {X 137.2836, Y 39.7516, Z -1.3333, A 0.000, B 0.000, C 0.000 }
gfCNCPoint1[4636] = {X 137.2836, Y 23.8768, Z -1.3333, A 0.000, B 0.000, C 0.000 }
gfCNCPoint1[4637] = {X 136.4352, Y 24.2641, Z -1.3333, A 0.000, B 0.000, C 0.000 }
gfCNCPoint1[4638] = {X 135.5443, Y 24.5398, Z -1.3333, A 0.000, B 0.000, C 0.000 }
gfCNCPoint1[4639] = {X 134.6254, Y 24.6993, Z -1.3333, A 0.000, B 0.000, C 0.000 }
gfCNCPoint1[4640] = {X 134.2595, Y 24.7296, Z -1.3333, A 0.000, B 0.000, C 0.000 }
gfCNCPoint1[4641] = {X 133.8926, Y 24.7414, Z -1.3333, A 0.000, B 0.000, C 0.000 }
gfCNCPoint1[4642] = {X 133.2006, Y 24.7415, Z -1.3333, A 0.000, B 0.000, C 0.000 }
gfCNCPoint1[4643] = {X 131.9919, Y 24.6405, Z -1.3333, A 0.000, B 0.000, C 0.000 }
gfCNCPoint1[4644] = {X 130.8166, Y 24.3401, Z -1.3333, A 0.000, B 0.000, C 0.000 }
gfCNCPoint1[4645] = {X 129.7076, Y 23.8488, Z -1.3333, A 0.000, B 0.000, C 0.000 }
gfCNCPoint1[4646] = {X 128.6956, Y 23.1802, Z -1.3333, A 0.000, B 0.000, C 0.000 }
gfCNCPoint1[4647] = {X 127.8086, Y 22.3527, Z -1.3333, A 0.000, B 0.000, C 0.000 }
gfCNCPoint1[4648] = {X 127.0713, Y 21.3895, Z -1.3333, A 0.000, B 0.000, C 0.000 }
gfCNCPoint1[4649] = {X 126.5041, Y 20.3173, Z -1.3333, A 0.000, B 0.000, C 0.000 }
gfCNCPoint1[4650] = {X 126.1229, Y 19.1658, Z -1.3333, A 0.000, B 0.000, C 0.000 }
gfCNCPoint1[4651] = {X 125.9382, Y 17.9669, Z -1.3333, A 0.000, B 0.000, C 0.000 }
gfCNCPoint1[4652] = {X 125.9250, Y 17.7144, Z -1.3333, A 0.000, B 0.000, C 0.000 }
gfCNCPoint1[4653] = {X 125.9206, Y 17.4615, Z -1.3333, A 0.000, B 0.000, C 0.000 }
gfCNCPoint1[4654] = {X 125.9206, Y 10.4835, Z -1.3333, A 0.000, B 0.000, C 0.000 }
gfCNCPoint1[4655] = {X 125.9372, Y 9.9932, Z -1.3333, A 0.000, B 0.000, C 0.000 }
gfCNCPoint1[4656] = {X 125.9867, Y 9.5051, Z -1.3333, A 0.000, B 0.000, C 0.000 }
gfCNCPoint1[4657] = {X 121.8687, Y 9.5051, Z -1.3333, A 0.000, B 0.000, C 0.000 }
gfCNCPoint1[4658] = {X 122.3091, Y 10.3411, Z -1.3333, A 0.000, B 0.000, C 0.000 }
gfCNCPoint1[4659] = {X 122.5801, Y 11.2463, Z -1.3333, A 0.000, B 0.000, C 0.000 }
gfCNCPoint1[4660] = {X 122.6716, Y 12.1868, Z -1.3333, A 0.000, B 0.000, C 0.000 }
gfCNCPoint1[4661] = {X 122.6714, Y 13.0237, Z -1.3333, A 0.000, B 0.000, C 0.000 }
gfCNCPoint1[4662] = {X 122.5640, Y 13.9972, Z -1.3333, A 0.000, B 0.000, C 0.000 }
gfCNCPoint1[4663] = {X 122.2644, Y 14.9295, Z -1.3333, A 0.000, B 0.000, C 0.000 }
gfCNCPoint1[4664] = {X 121.7846, Y 15.7833, Z -1.3333, A 0.000, B 0.000, C 0.000 }
gfCNCPoint1[4665] = {X 121.1441, Y 16.5242, Z -1.3333, A 0.000, B 0.000, C 0.000 }
gfCNCPoint1[4666] = {X 121.1429, Y 40.6615, Z -1.3333, A 0.000, B 0.000, C 0.000 }
gfCNCPoint1[4667] = {X 121.7847, Y 41.4036, Z -1.3333, A 0.000, B 0.000, C 0.000 }
gfCNCPoint1[4668] = {X 122.2652, Y 42.2591, Z -1.3333, A 0.000, B 0.000, C 0.000 }
gfCNCPoint1[4669] = {X 122.5648, Y 43.1934, Z -1.3333, A 0.000, B 0.000, C 0.000 }
gfCNCPoint1[4670] = {X 122.6714, Y 44.1688, Z -1.3333, A 0.000, B 0.000, C 0.000 }
gfCNCPoint1[4671] = {X 122.6716, Y 45.0000, Z -1.3333, A 0.000, B 0.000, C 0.000 }
gfCNCPoint1[4672] = {X 122.5778, Y 45.9520, Z -1.3333, A 0.000, B 0.000, C 0.000 }
gfCNCPoint1[4673] = {X 122.3001, Y 46.8675, Z -1.3333, A 0.000, B 0.000, C 0.000 }
gfCNCPoint1[4674] = {X 121.8491, Y 47.7112, Z -1.3333, A 0.000, B 0.000, C 0.000 }
gfCNCPoint1[4675] = {X 121.2423, Y 48.4507, Z -1.3333, A 0.000, B 0.000, C 0.000 }
gfCNCPoint1[4676] = {X 120.5028, Y 49.0576, Z -1.3333, A 0.000, B 0.000, C 0.000 }
gfCNCPoint1[4677] = {X 119.6591, Y 49.5085, Z -1.3333, A 0.000, B 0.000, C 0.000 }
gfCNCPoint1[4678] = {X 118.7436, Y 49.7862, Z -1.3333, A 0.000, B 0.000, C 0.000 }
gfCNCPoint1[4679] = {X 117.7916, Y 49.8800, Z -1.3333, A 0.000, B 0.000, C 0.000 }
gfCNCPoint1[4680] = {X 111.9185, Y 49.8800, Z -1.3333, A 0.000, B 0.000, C 0.000 }
gfCNCPoint1[4681] = {X 111.0234, Y 49.7972, Z -1.3333, A 0.000, B 0.000, C 0.000 }
gfCNCPoint1[4682] = {X 110.1587, Y 49.5517, Z -1.3333, A 0.000, B 0.000, C 0.000 }
gfCNCPoint1[4683] = {X 109.3537, Y 49.1517, Z -1.3333, A 0.000, B 0.000, C 0.000 }
gfCNCPoint1[4684] = {X 108.6357, Y 48.6108, Z -1.3333, A 0.000, B 0.000, C 0.000 }
gfCNCPoint1[4685] = {X 108.0714, Y 48.0024, Z -1.3333, A 0.000, B 0.000, C 0.000 }
gfCNCPoint1[4686] = {X 107.6183, Y 47.3071, Z -1.3333, A 0.000, B 0.000, C 0.000 }
gfCNCPoint1[4687] = {X 107.2895, Y 46.5451, Z -1.3333, A 0.000, B 0.000, C 0.000 }
gfCNCPoint1[4688] = {X 107.0947, Y 45.7384, Z -1.3333, A 0.000, B 0.000, C 0.000 }
gfCNCPoint1[4689] = {X 106.6287, Y 46.8768, Z -1.3333, A 0.000, B 0.000, C 0.000 }
gfCNCPoint1[4690] = {X 106.1131, Y 47.8110, Z -1.3333, A 0.000, B 0.000, C 0.000 }
gfCNCPoint1[4691] = {X 105.4068, Y 48.6108, Z -1.3333, A 0.000, B 0.000, C 0.000 }
gfCNCPoint1[4692] = {X 104.8391, Y 49.0550, Z -1.3333, A 0.000, B 0.000, C 0.000 }
gfCNCPoint1[4693] = {X 104.2121, Y 49.4107, Z -1.3333, A 0.000, B 0.000, C 0.000 }
gfCNCPoint1[4694] = {X 103.3106, Y 49.7335, Z -1.3333, A 0.000, B 0.000, C 0.000 }
gfCNCPoint1[4695] = {X 102.3635, Y 49.8741, Z -1.3333, A 0.000, B 0.000, C 0.000 }
gfCNCPoint1[4696] = {X 101.4071, Y 49.8271, Z -1.3333, A 0.000, B 0.000, C 0.000 }
gfCNCPoint1[4697] = {X 100.4784, Y 49.5941, Z -1.3333, A 0.000, B 0.000, C 0.000 }
gfCNCPoint1[4698] = {X 99.6130, Y 49.1844, Z -1.3333, A 0.000, B 0.000, C 0.000 }
gfCNCPoint1[4699] = {X 98.8443, Y 48.6135, Z -1.3333, A 0.000, B 0.000, C 0.000 }
gfCNCPoint1[4700] = {X 98.1362, Y 47.8127, Z -1.3333, A 0.000, B 0.000, C 0.000 }
gfCNCPoint1[4701] = {X 97.6194, Y 46.8769, Z -1.3333, A 0.000, B 0.000, C 0.000 }
gfCNCPoint1[4702] = {X 97.1600, Y 45.7536, Z -1.3333, A 0.000, B 0.000, C 0.000 }
gfCNCPoint1[4703] = {X 96.9635, Y 46.5570, Z -1.3333, A 0.000, B 0.000, C 0.000 }
gfCNCPoint1[4704] = {X 96.6342, Y 47.3156, Z -1.3333, A 0.000, B 0.000, C 0.000 }
gfCNCPoint1[4705] = {X 96.1814, Y 48.0078, Z -1.3333, A 0.000, B 0.000, C 0.000 }
gfCNCPoint1[4706] = {X 95.6183, Y 48.6135, Z -1.3333, A 0.000, B 0.000, C 0.000 }
gfCNCPoint1[4707] = {X 94.9007, Y 49.1533, Z -1.3333, A 0.000, B 0.000, C 0.000 }
gfCNCPoint1[4708] = {X 94.0964, Y 49.5524, Z -1.3333, A 0.000, B 0.000, C 0.000 }
gfCNCPoint1[4709] = {X 93.2326, Y 49.7974, Z -1.3333, A 0.000, B 0.000, C 0.000 }
gfCNCPoint1[4710] = {X 92.3385, Y 49.8800, Z -1.3333, A 0.000, B 0.000, C 0.000 }
gfCNCPoint1[4711] = {X 85.8951, Y 49.8800, Z -1.3333, A 0.000, B 0.000, C 0.000 }
gfCNCPoint1[4712] = {X 85.0841, Y 49.8121, Z -1.3333, A 0.000, B 0.000, C 0.000 }
gfCNCPoint1[4713] = {X 84.2956, Y 49.6104, Z -1.3333, A 0.000, B 0.000, C 0.000 }
gfCNCPoint1[4714] = {X 83.5517, Y 49.2805, Z -1.3333, A 0.000, B 0.000, C 0.000 }
gfCNCPoint1[4715] = {X 82.8729, Y 48.8316, Z -1.3333, A 0.000, B 0.000, C 0.000 }
gfCNCPoint1[4716] = {X 82.2391, Y 48.2324, Z -1.3333, A 0.000, B 0.000, C 0.000 }
gfCNCPoint1[4717] = {X 81.7221, Y 47.5300, Z -1.3333, A 0.000, B 0.000, C 0.000 }
gfCNCPoint1[4718] = {X 81.3384, Y 46.7467, Z -1.3333, A 0.000, B 0.000, C 0.000 }
gfCNCPoint1[4719] = {X 81.1002, Y 45.9077, Z -1.3333, A 0.000, B 0.000, C 0.000 }
gfCNCPoint1[4720] = {X 81.0152, Y 45.0397, Z -1.3333, A 0.000, B 0.000, C 0.000 }
gfCNCPoint1[4721] = {X 81.0151, Y 44.2030, Z -1.3333, A 0.000, B 0.000, C 0.000 }
gfCNCPoint1[4722] = {X 81.1207, Y 43.2196, Z -1.3333, A 0.000, B 0.000, C 0.000 }
gfCNCPoint1[4723] = {X 81.4199, Y 42.2770, Z -1.3333, A 0.000, B 0.000, C 0.000 }
gfCNCPoint1[4724] = {X 81.9007, Y 41.4127, Z -1.3333, A 0.000, B 0.000, C 0.000 }
gfCNCPoint1[4725] = {X 82.5440, Y 40.6615, Z -1.3333, A 0.000, B 0.000, C 0.000 }
gfCNCPoint1[4726] = {X 82.5437, Y 16.5252, Z -1.3333, A 0.000, B 0.000, C 0.000 }
gfCNCPoint1[4727] = {X 81.9021, Y 15.7835, Z -1.3333, A 0.000, B 0.000, C 0.000 }
gfCNCPoint1[4728] = {X 81.4218, Y 14.9284, Z -1.3333, A 0.000, B 0.000, C 0.000 }
gfCNCPoint1[4729] = {X 81.1221, Y 13.9945, Z -1.3333, A 0.000, B 0.000, C 0.000 }
gfCNCPoint1[4730] = {X 81.0153, Y 13.0196, Z -1.3333, A 0.000, B 0.000, C 0.000 }
gfCNCPoint1[4731] = {X 81.0151, Y 12.1868, Z -1.3333, A 0.000, B 0.000, C 0.000 }
gfCNCPoint1[4732] = {X 81.0160, Y 12.0924, Z -1.3333, A 0.000, B 0.000, C 0.000 }
gfCNCPoint1[4733] = {X 81.0187, Y 11.9980, Z -1.3333, A 0.000, B 0.000, C 0.000 }
gfCNCPoint1[4734] = {X 81.1324, Y 11.1231, Z -1.3333, A 0.000, B 0.000, C 0.000 }
gfCNCPoint1[4735] = {X 81.4018, Y 10.2830, Z -1.3333, A 0.000, B 0.000, C 0.000 }
gfCNCPoint1[4736] = {X 81.8180, Y 9.5051, Z -1.3333, A 0.000, B 0.000, C 0.000 }
gfCNCPoint1[4737] = {X 82.2190, Y 9.7689, Z -1.3333, A 0.000, B 0.000, C 0.000 }
gfCNCPoint1[4738] = {X 82.7658, Y 9.0936, Z -1.3333, A 0.000, B 0.000, C 0.000 }
gfCNCPoint1[4739] = {X 83.4347, Y 8.5390, Z -1.3333, A 0.000, B 0.000, C 0.000 }
gfCNCPoint1[4740] = {X 84.1995, Y 8.1266, Z -1.3333, A 0.000, B 0.000, C 0.000 }
gfCNCPoint1[4741] = {X 85.0304, Y 7.8726, Z -1.3333, A 0.000, B 0.000, C 0.000 }
gfCNCPoint1[4742] = {X 85.8951, Y 7.7868, Z -1.3333, A 0.000, B 0.000, C 0.000 }
gfCNCPoint1[4743] = {X 94.0497, Y 7.7868, Z -1.3333, A 0.000, B 0.000, C 0.000 }
gfCNCPoint1[4744] = {X 95.0288, Y 7.8971, Z -1.3333, A 0.000, B 0.000, C 0.000 }
gfCNCPoint1[4745] = {X 95.9588, Y 8.2226, Z -1.3333, A 0.000, B 0.000, C 0.000 }
gfCNCPoint1[4746] = {X 96.7930, Y 8.7468, Z -1.3333, A 0.000, B 0.000, C 0.000 }
gfCNCPoint1[4747] = {X 97.4897, Y 9.4435, Z -1.3333, A 0.000, B 0.000, C 0.000 }
gfCNCPoint1[4748] = {X 98.0139, Y 10.2777, Z -1.3333, A 0.000, B 0.000, C 0.000 }
gfCNCPoint1[4749] = {X 98.3394, Y 11.2077, Z -1.3333, A 0.000, B 0.000, C 0.000 }
gfCNCPoint1[4750] = {X 98.4497, Y 12.1868, Z -1.3333, A 0.000, B 0.000, C 0.000 }
gfCNCPoint1[4751] = {X 98.4494, Y 13.0233, Z -1.3333, A 0.000, B 0.000, C 0.000 }
gfCNCPoint1[4752] = {X 98.3723, Y 13.7996, Z -1.3333, A 0.000, B 0.000, C 0.000 }
gfCNCPoint1[4753] = {X 98.1592, Y 14.5501, Z -1.3333, A 0.000, B 0.000, C 0.000 }
gfCNCPoint1[4754] = {X 97.8170, Y 15.2512, Z -1.3333, A 0.000, B 0.000, C 0.000 }
gfCNCPoint1[4755] = {X 98.3666, Y 16.6194, Z -1.3333, A 0.000, B 0.000, C 0.000 }
gfCNCPoint1[4756] = {X 101.7170, Y 24.9264, Z -1.3333, A 0.000, B 0.000, C 0.000 }
gfCNCPoint1[4757] = {X 101.8768, Y 25.3192, Z -1.3333, A 0.000, B 0.000, C 0.000 }
gfCNCPoint1[4758] = {X 105.9248, Y 15.2241, Z -1.3333, A 0.000, B 0.000, C 0.000 }
gfCNCPoint1[4759] = {X 105.5859, Y 14.5163, Z -1.3333, A 0.000, B 0.000, C 0.000 }
gfCNCPoint1[4760] = {X 105.3782, Y 13.7595, Z -1.3333, A 0.000, B 0.000, C 0.000 }
gfCNCPoint1[4761] = {X 105.3083, Y 12.9779, Z -1.3333, A 0.000, B 0.000, C 0.000 }
gfCNCPoint1[4762] = {X 105.3083, Y 12.1868, Z -1.3333, A 0.000, B 0.000, C 0.000 }
gfCNCPoint1[4763] = {X 105.4186, Y 11.2077, Z -1.3333, A 0.000, B 0.000, C 0.000 }
gfCNCPoint1[4764] = {X 105.7440, Y 10.2777, Z -1.3333, A 0.000, B 0.000, C 0.000 }
gfCNCPoint1[4765] = {X 106.2682, Y 9.4435, Z -1.3333, A 0.000, B 0.000, C 0.000 }
gfCNCPoint1[4766] = {X 106.9649, Y 8.7468, Z -1.3333, A 0.000, B 0.000, C 0.000 }
gfCNCPoint1[4767] = {X 107.7992, Y 8.2226, Z -1.3333, A 0.000, B 0.000, C 0.000 }
gfCNCPoint1[4768] = {X 108.7292, Y 7.8971, Z -1.3333, A 0.000, B 0.000, C 0.000 }
gfCNCPoint1[4769] = {X 109.7083, Y 7.7868, Z -1.3333, A 0.000, B 0.000, C 0.000 }
gfCNCPoint1[4770] = {X 117.7916, Y 7.7868, Z -1.3333, A 0.000, B 0.000, C 0.000 }
gfCNCPoint1[4771] = {X 118.7707, Y 7.8971, Z -1.3333, A 0.000, B 0.000, C 0.000 }
gfCNCPoint1[4772] = {X 119.7007, Y 8.2226, Z -1.3333, A 0.000, B 0.000, C 0.000 }
gfCNCPoint1[4773] = {X 120.5349, Y 8.7468, Z -1.3333, A 0.000, B 0.000, C 0.000 }
gfCNCPoint1[4774] = {X 121.2316, Y 9.4435, Z -1.3333, A 0.000, B 0.000, C 0.000 }
gfCNCPoint1[4775] = {X 121.7558, Y 10.2777, Z -1.3333, A 0.000, B 0.000, C 0.000 }
gfCNCPoint1[4776] = {X 122.0813, Y 11.2077, Z -1.3333, A 0.000, B 0.000, C 0.000 }
gfCNCPoint1[4777] = {X 122.1916, Y 12.1868, Z -1.3333, A 0.000, B 0.000, C 0.000 }
gfCNCPoint1[4778] = {X 122.1913, Y 13.0233, Z -1.3333, A 0.000, B 0.000, C 0.000 }
gfCNCPoint1[4779] = {X 122.0830, Y 13.9493, Z -1.3333, A 0.000, B 0.000, C 0.000 }
gfCNCPoint1[4780] = {X 121.7820, Y 14.8317, Z -1.3333, A 0.000, B 0.000, C 0.000 }
gfCNCPoint1[4781] = {X 121.3019, Y 15.6309, Z -1.3333, A 0.000, B 0.000, C 0.000 }
gfCNCPoint1[4782] = {X 120.6641, Y 16.3110, Z -1.3333, A 0.000, B 0.000, C 0.000 }
gfCNCPoint1[4783] = {X 120.6628, Y 40.8753, Z -1.3333, A 0.000, B 0.000, C 0.000 }
gfCNCPoint1[4784] = {X 120.6784, Y 40.8882, Z -1.3333, A 0.000, B 0.000, C 0.000 }
gfCNCPoint1[4785] = {X 121.3172, Y 41.5764, Z -1.3333, A 0.000, B 0.000, C 0.000 }
gfCNCPoint1[4786] = {X 121.7955, Y 42.3843, Z -1.3333, A 0.000, B 0.000, C 0.000 }
gfCNCPoint1[4787] = {X 122.0914, Y 43.2754, Z -1.3333, A 0.000, B 0.000, C 0.000 }
gfCNCPoint1[4788] = {X 122.1916, Y 44.2089, Z -1.3333, A 0.000, B 0.000, C 0.000 }
gfCNCPoint1[4789] = {X 122.1916, Y 45.0000, Z -1.3333, A 0.000, B 0.000, C 0.000 }
gfCNCPoint1[4790] = {X 122.0813, Y 45.9791, Z -1.3333, A 0.000, B 0.000, C 0.000 }
gfCNCPoint1[4791] = {X 121.7558, Y 46.9091, Z -1.3333, A 0.000, B 0.000, C 0.000 }
gfCNCPoint1[4792] = {X 121.2316, Y 47.7434, Z -1.3333, A 0.000, B 0.000, C 0.000 }
gfCNCPoint1[4793] = {X 120.5349, Y 48.4401, Z -1.3333, A 0.000, B 0.000, C 0.000 }
gfCNCPoint1[4794] = {X 119.7007, Y 48.9643, Z -1.3333, A 0.000, B 0.000, C 0.000 }
gfCNCPoint1[4795] = {X 118.7707, Y 49.2897, Z -1.3333, A 0.000, B 0.000, C 0.000 }
gfCNCPoint1[4796] = {X 117.7916, Y 49.4000, Z -1.3333, A 0.000, B 0.000, C 0.000 }
gfCNCPoint1[4797] = {X 111.9185, Y 49.4000, Z -1.3333, A 0.000, B 0.000, C 0.000 }
gfCNCPoint1[4798] = {X 110.9394, Y 49.2897, Z -1.3333, A 0.000, B 0.000, C 0.000 }
gfCNCPoint1[4799] = {X 110.0094, Y 48.9643, Z -1.3333, A 0.000, B 0.000, C 0.000 }
gfCNCPoint1[4800] = {X 109.1751, Y 48.4400, Z -1.3333, A 0.000, B 0.000, C 0.000 }
gfCNCPoint1[4801] = {X 108.4784, Y 47.7433, Z -1.3333, A 0.000, B 0.000, C 0.000 }
gfCNCPoint1[4802] = {X 107.9542, Y 46.9091, Z -1.3333, A 0.000, B 0.000, C 0.000 }
gfCNCPoint1[4803] = {X 107.6288, Y 45.9790, Z -1.3333, A 0.000, B 0.000, C 0.000 }
gfCNCPoint1[4804] = {X 107.5185, Y 44.9999, Z -1.3333, A 0.000, B 0.000, C 0.000 }
gfCNCPoint1[4805] = {X 107.5185, Y 44.1795, Z -1.3333, A 0.000, B 0.000, C 0.000 }
gfCNCPoint1[4806] = {X 107.5551, Y 43.6246, Z -1.3333, A 0.000, B 0.000, C 0.000 }
gfCNCPoint1[4807] = {X 107.6642, Y 43.0792, Z -1.3333, A 0.000, B 0.000, C 0.000 }
gfCNCPoint1[4808] = {X 106.1856, Y 46.6923, Z -1.3333, A 0.000, B 0.000, C 0.000 }
gfCNCPoint1[4809] = {X 105.8087, Y 47.4049, Z -1.3333, A 0.000, B 0.000, C 0.000 }
gfCNCPoint1[4810] = {X 105.3081, Y 48.0367, Z -1.3333, A 0.000, B 0.000, C 0.000 }
gfCNCPoint1[4811] = {X 104.7006, Y 48.5667, Z -1.3333, A 0.000, B 0.000, C 0.000 }
gfCNCPoint1[4812] = {X 104.0067, Y 48.9769, Z -1.3333, A 0.000, B 0.000, C 0.000 }
gfCNCPoint1[4813] = {X 103.0414, Y 49.3033, Z -1.3333, A 0.000, B 0.000, C 0.000 }
gfCNCPoint1[4814] = {X 102.0269, Y 49.3989, Z -1.3333, A 0.000, B 0.000, C 0.000 }
gfCNCPoint1[4815] = {X 101.0176, Y 49.2586, Z -1.3333, A 0.000, B 0.000, C 0.000 }
gfCNCPoint1[4816] = {X 100.0676, Y 48.8899, Z -1.3333, A 0.000, B 0.000, C 0.000 }
gfCNCPoint1[4817] = {X 99.2280, Y 48.3125, Z -1.3333, A 0.000, B 0.000, C 0.000 }
gfCNCPoint1[4818] = {X 98.5436, Y 47.5575, Z -1.3333, A 0.000, B 0.000, C 0.000 }
gfCNCPoint1[4819] = {X 98.0514, Y 46.6653, Z -1.3333, A 0.000, B 0.000, C 0.000 }
gfCNCPoint1[4820] = {X 96.5848, Y 43.0786, Z -1.3333, A 0.000, B 0.000, C 0.000 }
gfCNCPoint1[4821] = {X 96.6977, Y 43.6389, Z -1.3333, A 0.000, B 0.000, C 0.000 }
gfCNCPoint1[4822] = {X 96.7385, Y 44.2089, Z -1.3333, A 0.000, B 0.000, C 0.000 }
gfCNCPoint1[4823] = {X 96.7383, Y 45.0423, Z -1.3333, A 0.000, B 0.000, C 0.000 }
gfCNCPoint1[4824] = {X 96.6200, Y 46.0144, Z -1.3333, A 0.000, B 0.000, C 0.000 }
gfCNCPoint1[4825] = {X 96.2896, Y 46.9363, Z -1.3333, A 0.000, B 0.000, C 0.000 }
gfCNCPoint1[4826] = {X 95.7635, Y 47.7622, Z -1.3333, A 0.000, B 0.000, C 0.000 }
gfCNCPoint1[4827] = {X 95.0677, Y 48.4513, Z -1.3333, A 0.000, B 0.000, C 0.000 }
gfCNCPoint1[4828] = {X 94.2367, Y 48.9695, Z -1.3333, A 0.000, B 0.000, C 0.000 }
gfCNCPoint1[4829] = {X 93.3117, Y 49.2910, Z -1.3333, A 0.000, B 0.000, C 0.000 }
gfCNCPoint1[4830] = {X 92.3385, Y 49.4000, Z -1.3333, A 0.000, B 0.000, C 0.000 }
gfCNCPoint1[4831] = {X 85.8951, Y 49.4000, Z -1.3333, A 0.000, B 0.000, C 0.000 }
gfCNCPoint1[4832] = {X 84.9160, Y 49.2897, Z -1.3333, A 0.000, B 0.000, C 0.000 }
gfCNCPoint1[4833] = {X 83.9860, Y 48.9643, Z -1.3333, A 0.000, B 0.000, C 0.000 }
gfCNCPoint1[4834] = {X 83.1517, Y 48.4400, Z -1.3333, A 0.000, B 0.000, C 0.000 }
gfCNCPoint1[4835] = {X 82.4550, Y 47.7433, Z -1.3333, A 0.000, B 0.000, C 0.000 }
gfCNCPoint1[4836] = {X 81.9308, Y 46.9091, Z -1.3333, A 0.000, B 0.000, C 0.000 }
gfCNCPoint1[4837] = {X 81.6054, Y 45.9791, Z -1.3333, A 0.000, B 0.000, C 0.000 }
gfCNCPoint1[4838] = {X 81.4951, Y 45.0000, Z -1.3333, A 0.000, B 0.000, C 0.000 }
gfCNCPoint1[4839] = {X 81.4951, Y 44.2062, Z -1.3333, A 0.000, B 0.000, C 0.000 }
gfCNCPoint1[4840] = {X 81.6010, Y 43.2692, Z -1.3333, A 0.000, B 0.000, C 0.000 }
gfCNCPoint1[4841] = {X 81.9015, Y 42.3754, Z -1.3333, A 0.000, B 0.000, C 0.000 }
gfCNCPoint1[4842] = {X 82.3829, Y 41.5646, Z -1.3333, A 0.000, B 0.000, C 0.000 }
